LIN {X 0,Y 438.621,Z 496.858,A -85,B 0,C 180,E1 -9202.616,E2 -9202.616} C_VEL
LIN {X 0,Y 438.766,Z 492.887,A -85,B 0,C 180,E1 -9205.625,E2 -9205.625} C_VEL
LIN {X 0,Y 438.907,Z 491.24,A -85,B 0,C 180,E1 -9206.895,E2 -9206.895} C_VEL
LIN {X 0,Y 439.036,Z 496.514,A -85,B 0,C 180,E1 -9209.225,E2 -9209.225} C_VEL
LIN {X 0,Y 438.959,Z 503.716,A -85,B 0,C 180,E1 -9212.435,E2 -9212.435} C_VEL
LIN {X 0,Y 438.851,Z 509.893,A -85,B 0,C 180,E1 -9215.239,E2 -9215.239} C_VEL
LIN {X 0,Y 438.736,Z 517.378,A -85,B 0,C 180,E1 -9218.663,E2 -9218.663} C_VEL
LIN {X 0,Y 438.606,Z 523.965,A -85,B 0,C 180,E1 -9221.684,E2 -9221.684} C_VEL
LIN {X 0,Y 438.602,Z 527.103,A -85,B 0,C 180,E1 -9223.131,E2 -9223.131} C_VEL
LIN {X 0,Y 440.498,Z 538.596,A -85,B 0,C 180,E1 -9223.601,E2 -9223.601} C_VEL
LIN {X 0,Y 441.012,Z 543.733,A -85,B 0,C 180,E1 -9223.868,E2 -9223.868} C_VEL
LIN {X 0,Y 440.734,Z 552.93,A -85,B 0,C 180,E1 -9224.41,E2 -9224.41} C_VEL
LIN {X 0,Y 440.34,Z 561.813,A -85,B 0,C 180,E1 -9225.077,E2 -9225.077} C_VEL
LIN {X 0,Y 439.852,Z 572.155,A -85,B 0,C 180,E1 -9226.085,E2 -9226.085} C_VEL
LIN {X 0,Y 439.464,Z 579.635,A -85,B 0,C 180,E1 -9227.014,E2 -9227.014} C_VEL
LIN {X 0,Y 439.174,Z 584.756,A -85,B 0,C 180,E1 -9227.769,E2 -9227.769} C_VEL
LIN {X 0,Y 438.86,Z 590.657,A -85,B 0,C 180,E1 -9228.822,E2 -9228.822} C_VEL
LIN {X 0,Y 438.691,Z 595.327,A -85,B 0,C 180,E1 -9229.847,E2 -9229.847} C_VEL
LIN {X 0,Y 438.469,Z 600.506,A -85,B 0,C 180,E1 -9231.309,E2 -9231.309} C_VEL
LIN {X 0,Y 438.381,Z 603.477,A -85,B 0,C 180,E1 -9232.467,E2 -9232.467} C_VEL
LIN {X 0,Y 438.266,Z 605.527,A -85,B 0,C 180,E1 -9233.606,E2 -9233.606} C_VEL
LIN {X 0,Y 438.17,Z 606.89,A -85,B 0,C 180,E1 -9234.886,E2 -9234.886} C_VEL
LIN {X 0,Y 438.14,Z 607.23,A -85,B 0,C 180,E1 -9235.846,E2 -9235.846} C_VEL
LIN {X 0,Y 438.122,Z 606.973,A -85,B 0,C 180,E1 -9236.947,E2 -9236.947} C_VEL
LIN {X 0,Y 438.231,Z 605.831,A -85,B 0,C 180,E1 -9238.209,E2 -9238.209} C_VEL
LIN {X 0,Y 438.323,Z 604.322,A -85,B 0,C 180,E1 -9239.13,E2 -9239.13} C_VEL
LIN {X 0,Y 438.443,Z 600.496,A -85,B 0,C 180,E1 -9240.731,E2 -9240.731} C_VEL
LIN {X 0,Y 438.648,Z 595.849,A -85,B 0,C 180,E1 -9242.059,E2 -9242.059} C_VEL
LIN {X 0,Y 438.883,Z 591.19,A -85,B 0,C 180,E1 -9243.103,E2 -9243.103} C_VEL
LIN {X 0,Y 439.181,Z 584.982,A -85,B 0,C 180,E1 -9244.227,E2 -9244.227} C_VEL
LIN {X 0,Y 439.567,Z 576.57,A -85,B 0,C 180,E1 -9245.436,E2 -9245.436} C_VEL
LIN {X 0,Y 439.972,Z 568.448,A -85,B 0,C 180,E1 -9246.344,E2 -9246.344} C_VEL
LIN {X 0,Y 440.298,Z 560.08,A -85,B 0,C 180,E1 -9247.103,E2 -9247.103} C_VEL
LIN {X 0,Y 440.718,Z 550.964,A -85,B 0,C 180,E1 -9247.759,E2 -9247.759} C_VEL
LIN {X 0,Y 440.817,Z 542.35,A -85,B 0,C 180,E1 -9248.249,E2 -9248.249} C_VEL
LIN {X 0,Y 438.98,Z 530.4,A -85,B 0,C 180,E1 -9248.794,E2 -9248.794} C_VEL
LIN {X 0,Y 438.451,Z 527.192,A -85,B 0,C 180,E1 -9248.921,E2 -9248.921} C_VEL
LIN {X 0,Y 438.501,Z 521.905,A -85,B 0,C 180,E1 -9251.539,E2 -9251.539} C_VEL
LIN {X 0,Y 438.633,Z 516.526,A -85,B 0,C 180,E1 -9254.193,E2 -9254.193} C_VEL
LIN {X 0,Y 438.625,Z 514.073,A -85,B 0,C 180,E1 -9255.408,E2 -9255.408} C_VEL
LIN {X 0,Y 437.974,Z 512.647,A -85,B 0,C 180,E1 -9256.152,E2 -9256.152} C_VEL
LIN {X 0,Y 435.187,Z 510.501,A -85,B 0,C 180,E1 -9257.368,E2 -9257.368} C_VEL
LIN {X 0,Y 432.835,Z 508.797,A -85,B 0,C 180,E1 -9258.35,E2 -9258.35} C_VEL
LIN {X 0,Y 431.834,Z 507.335,A -85,B 0,C 180,E1 -9259.103,E2 -9259.103} C_VEL
LIN {X 0,Y 431.757,Z 506.816,A -85,B 0,C 180,E1 -9259.357,E2 -9259.357} C_VEL
LIN {X 0,Y 431.93,Z 499.414,A -85,B 0,C 180,E1 -9262.998,E2 -9262.998} C_VEL
LIN {X 0,Y 432.055,Z 494.709,A -85,B 0,C 180,E1 -9265.334,E2 -9265.334} C_VEL
LIN {X 0,Y 432.018,Z 491.487,A -85,B 0,C 180,E1 -9266.969,E2 -9266.969} C_VEL
LIN {X 0,Y 432.524,Z 491.421,A -85,B 0,C 180,E1 -9269.068,E2 -9269.068} C_VEL
LIN {X 0,Y 432.727,Z 491.397,A -85,B 0,C 180,E1 -9270,E2 -9270} C_VEL
LIN {X 0,Y 432.606,Z 491.412,A -85,B 0,C 180,E1 -9272.793,E2 -9272.793} C_VEL
LIN {X 0,Y 432.575,Z 491.416,A -85,B 0,C 180,E1 -9276.53,E2 -9276.53} C_VEL
LIN {X 0,Y 432.443,Z 491.429,A -85,B 0,C 180,E1 -9279.353,E2 -9279.353} C_VEL
LIN {X 0,Y 432.432,Z 491.432,A -85,B 0,C 180,E1 -9282.803,E2 -9282.803} C_VEL
LIN {X 0,Y 432.413,Z 491.436,A -85,B 0,C 180,E1 -9286.478,E2 -9286.478} C_VEL
LIN {X 0,Y 432.34,Z 491.445,A -85,B 0,C 180,E1 -9289.96,E2 -9289.96} C_VEL
LIN {X 0,Y 432.32,Z 491.446,A -85,B 0,C 180,E1 -9292.964,E2 -9292.964} C_VEL
LIN {X 0,Y 432.365,Z 491.442,A -85,B 0,C 180,E1 -9296.032,E2 -9296.032} C_VEL
LIN {X 0,Y 432.352,Z 491.441,A -85,B 0,C 180,E1 -9299.186,E2 -9299.186} C_VEL
LIN {X 0,Y 432.325,Z 491.449,A -85,B 0,C 180,E1 -9302.293,E2 -9302.293} C_VEL
LIN {X 0,Y 432.34,Z 491.444,A -85,B 0,C 180,E1 -9304.676,E2 -9304.676} C_VEL
LIN {X 0,Y 432.346,Z 491.445,A -85,B 0,C 180,E1 -9308.148,E2 -9308.148} C_VEL
LIN {X 0,Y 432.333,Z 491.445,A -85,B 0,C 180,E1 -9311.602,E2 -9311.602} C_VEL
LIN {X 0,Y 432.34,Z 491.445,A -85,B 0,C 180,E1 -9314.346,E2 -9314.346} C_VEL
LIN {X 0,Y 432.364,Z 491.439,A -85,B 0,C 180,E1 -9317.009,E2 -9317.009} C_VEL
LIN {X 0,Y 432.356,Z 491.443,A -85,B 0,C 180,E1 -9319.816,E2 -9319.816} C_VEL
LIN {X 0,Y 432.314,Z 491.445,A -85,B 0,C 180,E1 -9323.023,E2 -9323.023} C_VEL
LIN {X 0,Y 432.357,Z 491.445,A -85,B 0,C 180,E1 -9325.996,E2 -9325.996} C_VEL
LIN {X 0,Y 432.345,Z 491.443,A -85,B 0,C 180,E1 -9329.489,E2 -9329.489} C_VEL
LIN {X 0,Y 432.391,Z 491.437,A -85,B 0,C 180,E1 -9332.928,E2 -9332.928} C_VEL
LIN {X 0,Y 432.369,Z 491.442,A -85,B 0,C 180,E1 -9336.023,E2 -9336.023} C_VEL
LIN {X 0,Y 432.348,Z 491.442,A -85,B 0,C 180,E1 -9339.046,E2 -9339.046} C_VEL
LIN {X 0,Y 432.376,Z 491.441,A -85,B 0,C 180,E1 -9342.011,E2 -9342.011} C_VEL
LIN {X 0,Y 432.393,Z 491.437,A -85,B 0,C 180,E1 -9344.926,E2 -9344.926} C_VEL
LIN {X 0,Y 432.478,Z 491.428,A -85,B 0,C 180,E1 -9347.804,E2 -9347.804} C_VEL
LIN {X 0,Y 432.49,Z 491.426,A -85,B 0,C 180,E1 -9351.59,E2 -9351.59} C_VEL
LIN {X 0,Y 432.595,Z 491.412,A -85,B 0,C 180,E1 -9354.406,E2 -9354.406} C_VEL
LIN {X 0,Y 432.604,Z 491.412,A -85,B 0,C 180,E1 -9358.138,E2 -9358.138} C_VEL
LIN {X 0,Y 432.731,Z 491.397,A -85,B 0,C 180,E1 -9360,E2 -9360} C_VEL
LIN {X 0,Y 432.604,Z 491.41,A -85,B 0,C 180,E1 -9362.793,E2 -9362.793} C_VEL
LIN {X 0,Y 432.571,Z 491.414,A -85,B 0,C 180,E1 -9366.53,E2 -9366.53} C_VEL
LIN {X 0,Y 432.441,Z 491.432,A -85,B 0,C 180,E1 -9369.353,E2 -9369.353} C_VEL
LIN {X 0,Y 432.428,Z 491.431,A -85,B 0,C 180,E1 -9372.804,E2 -9372.804} C_VEL
LIN {X 0,Y 432.41,Z 491.435,A -85,B 0,C 180,E1 -9376.479,E2 -9376.479} C_VEL
LIN {X 0,Y 432.336,Z 491.446,A -85,B 0,C 180,E1 -9379.96,E2 -9379.96} C_VEL
LIN {X 0,Y 432.317,Z 491.447,A -85,B 0,C 180,E1 -9382.964,E2 -9382.964} C_VEL
LIN {X 0,Y 432.362,Z 491.443,A -85,B 0,C 180,E1 -9386.033,E2 -9386.033} C_VEL
LIN {X 0,Y 432.35,Z 491.444,A -85,B 0,C 180,E1 -9389.187,E2 -9389.187} C_VEL
LIN {X 0,Y 432.329,Z 491.445,A -85,B 0,C 180,E1 -9392.295,E2 -9392.295} C_VEL
LIN {X 0,Y 432.338,Z 491.444,A -85,B 0,C 180,E1 -9394.677,E2 -9394.677} C_VEL
LIN {X 0,Y 432.344,Z 491.443,A -85,B 0,C 180,E1 -9398.149,E2 -9398.149} C_VEL
LIN {X 0,Y 432.332,Z 491.448,A -85,B 0,C 180,E1 -9401.603,E2 -9401.603} C_VEL
LIN {X 0,Y 432.338,Z 491.443,A -85,B 0,C 180,E1 -9404.347,E2 -9404.347} C_VEL
LIN {X 0,Y 432.318,Z 491.447,A -85,B 0,C 180,E1 -9407.016,E2 -9407.016} C_VEL
LIN {X 0,Y 432.355,Z 491.443,A -85,B 0,C 180,E1 -9409.817,E2 -9409.817} C_VEL
LIN {X 0,Y 432.316,Z 491.449,A -85,B 0,C 180,E1 -9413.024,E2 -9413.024} C_VEL
LIN {X 0,Y 432.398,Z 491.49,A -85,B 0,C 180,E1 -9414.446,E2 -9414.446} C_VEL
LIN {X 0,Y 433.697,Z 498.9,A -85,B 0,C 180,E1 -9417.673,E2 -9417.673} C_VEL
LIN {X 0,Y 433.795,Z 502.505,A -85,B 0,C 180,E1 -9419.167,E2 -9419.167} C_VEL
LIN {X 0,Y 433.235,Z 510.767,A -85,B 0,C 180,E1 -9422.463,E2 -9422.463} C_VEL
LIN {X 0,Y 432.665,Z 519.988,A -85,B 0,C 180,E1 -9426.041,E2 -9426.041} C_VEL
LIN {X 0,Y 432.198,Z 529.205,A -85,B 0,C 180,E1 -9429.537,E2 -9429.537} C_VEL
LIN {X 0,Y 431.798,Z 538.416,A -85,B 0,C 180,E1 -9432.965,E2 -9432.965} C_VEL
LIN {X 0,Y 431.544,Z 547.609,A -85,B 0,C 180,E1 -9436.342,E2 -9436.342} C_VEL
LIN {X 0,Y 431.538,Z 549.403,A -85,B 0,C 180,E1 -9436.997,E2 -9436.997} C_VEL
LIN {X 0,Y 432.951,Z 563.611,A -85,B 0,C 180,E1 -9437.595,E2 -9437.595} C_VEL
LIN {X 0,Y 433.462,Z 570.117,A -85,B 0,C 180,E1 -9437.951,E2 -9437.951} C_VEL
LIN {X 0,Y 433.093,Z 580.396,A -85,B 0,C 180,E1 -9438.653,E2 -9438.653} C_VEL
LIN {X 0,Y 432.629,Z 589.892,A -85,B 0,C 180,E1 -9439.47,E2 -9439.47} C_VEL
LIN {X 0,Y 432.228,Z 598.533,A -85,B 0,C 180,E1 -9440.407,E2 -9440.407} C_VEL
LIN {X 0,Y 431.857,Z 607.082,A -85,B 0,C 180,E1 -9441.578,E2 -9441.578} C_VEL
LIN {X 0,Y 431.625,Z 613.803,A -85,B 0,C 180,E1 -9442.751,E2 -9442.751} C_VEL
LIN {X 0,Y 431.392,Z 618.953,A -85,B 0,C 180,E1 -9443.881,E2 -9443.881} C_VEL
LIN {X 0,Y 431.312,Z 623.981,A -85,B 0,C 180,E1 -9445.327,E2 -9445.327} C_VEL
LIN {X 0,Y 431.253,Z 626.448,A -85,B 0,C 180,E1 -9446.263,E2 -9446.263} C_VEL
LIN {X 0,Y 431.315,Z 628.342,A -85,B 0,C 180,E1 -9447.199,E2 -9447.199} C_VEL
LIN {X 0,Y 431.241,Z 629.637,A -85,B 0,C 180,E1 -9448.133,E2 -9448.133} C_VEL
LIN {X 0,Y 431.217,Z 630.481,A -85,B 0,C 180,E1 -9449.067,E2 -9449.067} C_VEL
LIN {X 0,Y 431.229,Z 630.751,A -85,B 0,C 180,E1 -9450,E2 -9450} C_VEL
LIN {X 0,Y 431.217,Z 630.501,A -85,B 0,C 180,E1 -9450.934,E2 -9450.934} C_VEL
LIN {X 0,Y 431.241,Z 629.661,A -85,B 0,C 180,E1 -9451.868,E2 -9451.868} C_VEL
LIN {X 0,Y 431.298,Z 628.374,A -85,B 0,C 180,E1 -9452.802,E2 -9452.802} C_VEL
LIN {X 0,Y 431.258,Z 625.37,A -85,B 0,C 180,E1 -9454.206,E2 -9454.206} C_VEL
LIN {X 0,Y 431.381,Z 621.08,A -85,B 0,C 180,E1 -9455.61,E2 -9455.61} C_VEL
LIN {X 0,Y 431.574,Z 615.227,A -85,B 0,C 180,E1 -9457.016,E2 -9457.016} C_VEL
LIN {X 0,Y 431.798,Z 608.9,A -85,B 0,C 180,E1 -9458.188,E2 -9458.188} C_VEL
LIN {X 0,Y 432.103,Z 602.762,A -85,B 0,C 180,E1 -9459.125,E2 -9459.125} C_VEL
LIN {X 0,Y 432.504,Z 595.348,A -85,B 0,C 180,E1 -9460.061,E2 -9460.061} C_VEL
LIN {X 0,Y 432.877,Z 587.491,A -85,B 0,C 180,E1 -9460.88,E2 -9460.88} C_VEL
LIN {X 0,Y 433.315,Z 579.319,A -85,B 0,C 180,E1 -9461.579,E2 -9461.579} C_VEL
LIN {X 0,Y 433.54,Z 569.525,A -85,B 0,C 180,E1 -9462.261,E2 -9462.261} C_VEL
LIN {X 0,Y 432.645,Z 557.327,A -85,B 0,C 180,E1 -9462.928,E2 -9462.928} C_VEL
LIN {X 0,Y 431.458,Z 548.071,A -85,B 0,C 180,E1 -9463.332,E2 -9463.332} C_VEL
LIN {X 0,Y 431.671,Z 539.83,A -85,B 0,C 180,E1 -9466.506,E2 -9466.506} C_VEL
LIN {X 0,Y 431.98,Z 531.096,A -85,B 0,C 180,E1 -9469.978,E2 -9469.978} C_VEL
LIN {X 0,Y 432.36,Z 522.72,A -85,B 0,C 180,E1 -9473.469,E2 -9473.469} C_VEL
LIN {X 0,Y 432.861,Z 515.354,A -85,B 0,C 180,E1 -9476.749,E2 -9476.749} C_VEL
LIN {X 0,Y 433.501,Z 508.305,A -85,B 0,C 180,E1 -9480.171,E2 -9480.171} C_VEL
LIN {X 0,Y 433.965,Z 503.76,A -85,B 0,C 180,E1 -9482.634,E2 -9482.634} C_VEL
LIN {X 0,Y 433.895,Z 500.697,A -85,B 0,C 180,E1 -9484.536,E2 -9484.536} C_VEL
LIN {X 0,Y 433.311,Z 496.888,A -85,B 0,C 180,E1 -9487.369,E2 -9487.369} C_VEL
LIN {X 0,Y 432.757,Z 493.7,A -85,B 0,C 180,E1 -9490.512,E2 -9490.512} C_VEL
LIN {X 0,Y 432.395,Z 491.961,A -85,B 0,C 180,E1 -9493.052,E2 -9493.052} C_VEL
LIN {X 0,Y 432.336,Z 491.447,A -85,B 0,C 180,E1 -9494.348,E2 -9494.348} C_VEL
LIN {X 0,Y 432.327,Z 491.448,A -85,B 0,C 180,E1 -9497.015,E2 -9497.015} C_VEL
LIN {X 0,Y 432.339,Z 491.446,A -85,B 0,C 180,E1 -9499.821,E2 -9499.821} C_VEL
LIN {X 0,Y 432.325,Z 491.563,A -85,B 0,C 180,E1 -9502.803,E2 -9502.803} C_VEL
LIN {X 0,Y 432.584,Z 493.097,A -85,B 0,C 180,E1 -9505.953,E2 -9505.953} C_VEL
LIN {X 0,Y 432.57,Z 494.889,A -85,B 0,C 180,E1 -9508.674,E2 -9508.674} C_VEL
LIN {X 0,Y 432.324,Z 497.455,A -85,B 0,C 180,E1 -9511.873,E2 -9511.873} C_VEL
LIN {X 0,Y 432.05,Z 500.247,A -85,B 0,C 180,E1 -9514.98,E2 -9514.98} C_VEL
LIN {X 0,Y 431.887,Z 503.238,A -85,B 0,C 180,E1 -9518.057,E2 -9518.057} C_VEL
LIN {X 0,Y 431.798,Z 506.271,A -85,B 0,C 180,E1 -9521.003,E2 -9521.003} C_VEL
LIN {X 0,Y 431.694,Z 509.44,A -85,B 0,C 180,E1 -9523.933,E2 -9523.933} C_VEL
LIN {X 0,Y 431.578,Z 512.837,A -85,B 0,C 180,E1 -9526.822,E2 -9526.822} C_VEL
LIN {X 0,Y 433.76,Z 522.586,A -85,B 0,C 180,E1 -9527.335,E2 -9527.335} C_VEL
LIN {X 0,Y 434.354,Z 528.796,A -85,B 0,C 180,E1 -9527.7,E2 -9527.7} C_VEL
LIN {X 0,Y 433.88,Z 539.519,A -85,B 0,C 180,E1 -9528.437,E2 -9528.437} C_VEL
LIN {X 0,Y 433.496,Z 547.554,A -85,B 0,C 180,E1 -9529.137,E2 -9529.137} C_VEL
LIN {X 0,Y 433.088,Z 555.269,A -85,B 0,C 180,E1 -9529.954,E2 -9529.954} C_VEL
LIN {X 0,Y 432.727,Z 562.542,A -85,B 0,C 180,E1 -9530.889,E2 -9530.889} C_VEL
LIN {X 0,Y 432.281,Z 569.949,A -85,B 0,C 180,E1 -9532.057,E2 -9532.057} C_VEL
LIN {X 0,Y 432.003,Z 576.748,A -85,B 0,C 180,E1 -9533.461,E2 -9533.461} C_VEL
LIN {X 0,Y 431.62,Z 580.395,A -85,B 0,C 180,E1 -9534.394,E2 -9534.394} C_VEL
LIN {X 0,Y 431.678,Z 583.344,A -85,B 0,C 180,E1 -9535.331,E2 -9535.331} C_VEL
LIN {X 0,Y 431.528,Z 585.637,A -85,B 0,C 180,E1 -9536.265,E2 -9536.265} C_VEL
LIN {X 0,Y 431.393,Z 587.351,A -85,B 0,C 180,E1 -9537.199,E2 -9537.199} C_VEL
LIN {X 0,Y 431.332,Z 588.555,A -85,B 0,C 180,E1 -9538.133,E2 -9538.133} C_VEL
LIN {X 0,Y 431.25,Z 589.276,A -85,B 0,C 180,E1 -9539.066,E2 -9539.066} C_VEL
LIN {X 0,Y 431.231,Z 589.505,A -85,B 0,C 180,E1 -9540,E2 -9540} C_VEL
LIN {X 0,Y 431.235,Z 589.141,A -85,B 0,C 180,E1 -9540.934,E2 -9540.934} C_VEL
LIN {X 0,Y 431.295,Z 588.253,A -85,B 0,C 180,E1 -9541.868,E2 -9541.868} C_VEL
LIN {X 0,Y 431.379,Z 586.874,A -85,B 0,C 180,E1 -9542.802,E2 -9542.802} C_VEL
LIN {X 0,Y 431.522,Z 583.791,A -85,B 0,C 180,E1 -9544.203,E2 -9544.203} C_VEL
LIN {X 0,Y 431.604,Z 579.415,A -85,B 0,C 180,E1 -9545.607,E2 -9545.607} C_VEL
LIN {X 0,Y 431.963,Z 574.673,A -85,B 0,C 180,E1 -9546.744,E2 -9546.744} C_VEL
LIN {X 0,Y 432.077,Z 568.326,A -85,B 0,C 180,E1 -9547.947,E2 -9547.947} C_VEL
LIN {X 0,Y 432.369,Z 562.276,A -85,B 0,C 180,E1 -9548.883,E2 -9548.883} C_VEL
LIN {X 0,Y 432.776,Z 553.923,A -85,B 0,C 180,E1 -9549.936,E2 -9549.936} C_VEL
LIN {X 0,Y 433.224,Z 544.72,A -85,B 0,C 180,E1 -9550.87,E2 -9550.87} C_VEL
LIN {X 0,Y 433.664,Z 534.251,A -85,B 0,C 180,E1 -9551.688,E2 -9551.688} C_VEL
LIN {X 0,Y 433.847,Z 525.581,A -85,B 0,C 180,E1 -9552.217,E2 -9552.217} C_VEL
LIN {X 0,Y 432.406,Z 516.149,A -85,B 0,C 180,E1 -9552.701,E2 -9552.701} C_VEL
LIN {X 0,Y 431.403,Z 510.563,A -85,B 0,C 180,E1 -9552.962,E2 -9552.962} C_VEL
LIN {X 0,Y 431.44,Z 506.27,A -85,B 0,C 180,E1 -9556.077,E2 -9556.077} C_VEL
LIN {X 0,Y 431.505,Z 502.098,A -85,B 0,C 180,E1 -9559.15,E2 -9559.15} C_VEL
LIN {X 0,Y 431.528,Z 498.31,A -85,B 0,C 180,E1 -9561.999,E2 -9561.999} C_VEL
LIN {X 0,Y 431.662,Z 494.317,A -85,B 0,C 180,E1 -9565.044,E2 -9565.044} C_VEL
LIN {X 0,Y 431.851,Z 492.008,A -85,B 0,C 180,E1 -9566.826,E2 -9566.826} C_VEL
LIN {X 0,Y 432.009,Z 495.847,A -85,B 0,C 180,E1 -9568.539,E2 -9568.539} C_VEL
LIN {X 0,Y 431.937,Z 502.183,A -85,B 0,C 180,E1 -9571.377,E2 -9571.377} C_VEL
LIN {X 0,Y 431.896,Z 507.785,A -85,B 0,C 180,E1 -9573.911,E2 -9573.911} C_VEL
LIN {X 0,Y 431.732,Z 514.698,A -85,B 0,C 180,E1 -9577.093,E2 -9577.093} C_VEL
LIN {X 0,Y 431.6,Z 521.116,A -85,B 0,C 180,E1 -9580.063,E2 -9580.063} C_VEL
LIN {X 0,Y 431.558,Z 527.411,A -85,B 0,C 180,E1 -9582.921,E2 -9582.921} C_VEL
LIN {X 0,Y 433.185,Z 537.127,A -85,B 0,C 180,E1 -9583.312,E2 -9583.312} C_VEL
LIN {X 0,Y 434.092,Z 544.931,A -85,B 0,C 180,E1 -9583.719,E2 -9583.719} C_VEL
LIN {X 0,Y 433.645,Z 556.12,A -85,B 0,C 180,E1 -9584.416,E2 -9584.416} C_VEL
LIN {X 0,Y 433.215,Z 565.628,A -85,B 0,C 180,E1 -9585.222,E2 -9585.222} C_VEL
LIN {X 0,Y 432.802,Z 573.348,A -85,B 0,C 180,E1 -9586.037,E2 -9586.037} C_VEL
LIN {X 0,Y 432.436,Z 580.464,A -85,B 0,C 180,E1 -9586.953,E2 -9586.953} C_VEL
LIN {X 0,Y 431.99,Z 588.079,A -85,B 0,C 180,E1 -9588.162,E2 -9588.162} C_VEL
LIN {X 0,Y 431.705,Z 594.036,A -85,B 0,C 180,E1 -9589.368,E2 -9589.368} C_VEL
LIN {X 0,Y 431.517,Z 598.612,A -85,B 0,C 180,E1 -9590.566,E2 -9590.566} C_VEL
LIN {X 0,Y 431.335,Z 602.092,A -85,B 0,C 180,E1 -9591.745,E2 -9591.745} C_VEL
LIN {X 0,Y 431.222,Z 604.77,A -85,B 0,C 180,E1 -9592.996,E2 -9592.996} C_VEL
LIN {X 0,Y 431.093,Z 606.849,A -85,B 0,C 180,E1 -9594.601,E2 -9594.601} C_VEL
LIN {X 0,Y 431.026,Z 607.379,A -85,B 0,C 180,E1 -9596.332,E2 -9596.332} C_VEL
LIN {X 0,Y 431.102,Z 606.298,A -85,B 0,C 180,E1 -9597.965,E2 -9597.965} C_VEL
LIN {X 0,Y 431.16,Z 605.558,A -85,B 0,C 180,E1 -9598.559,E2 -9598.559} C_VEL
LIN {X 0,Y 431.275,Z 603.398,A -85,B 0,C 180,E1 -9599.732,E2 -9599.732} C_VEL
LIN {X 0,Y 431.361,Z 600.878,A -85,B 0,C 180,E1 -9600.739,E2 -9600.739} C_VEL
LIN {X 0,Y 431.585,Z 596.296,A -85,B 0,C 180,E1 -9602.084,E2 -9602.084} C_VEL
LIN {X 0,Y 431.814,Z 591.248,A -85,B 0,C 180,E1 -9603.237,E2 -9603.237} C_VEL
LIN {X 0,Y 432.11,Z 586.005,A -85,B 0,C 180,E1 -9604.21,E2 -9604.21} C_VEL
LIN {X 0,Y 432.426,Z 578.906,A -85,B 0,C 180,E1 -9605.29,E2 -9605.29} C_VEL
LIN {X 0,Y 432.948,Z 569.283,A -85,B 0,C 180,E1 -9606.438,E2 -9606.438} C_VEL
LIN {X 0,Y 433.311,Z 560.916,A -85,B 0,C 180,E1 -9607.22,E2 -9607.22} C_VEL
LIN {X 0,Y 433.709,Z 552.639,A -85,B 0,C 180,E1 -9607.841,E2 -9607.841} C_VEL
LIN {X 0,Y 433.9,Z 543.655,A -85,B 0,C 180,E1 -9608.377,E2 -9608.377} C_VEL
LIN {X 0,Y 432.458,Z 533.788,A -85,B 0,C 180,E1 -9608.864,E2 -9608.864} C_VEL
LIN {X 0,Y 431.377,Z 527.349,A -85,B 0,C 180,E1 -9609.121,E2 -9609.121} C_VEL
LIN {X 0,Y 431.429,Z 521.633,A -85,B 0,C 180,E1 -9611.97,E2 -9611.97} C_VEL
LIN {X 0,Y 431.55,Z 515.753,A -85,B 0,C 180,E1 -9614.896,E2 -9614.896} C_VEL
LIN {X 0,Y 431.753,Z 510.04,A -85,B 0,C 180,E1 -9617.783,E2 -9617.783} C_VEL
LIN {X 0,Y 431.757,Z 506.816,A -85,B 0,C 180,E1 -9619.357,E2 -9619.357} C_VEL
LIN {X 0,Y 431.118,Z 505.356,A -85,B 0,C 180,E1 -9620.111,E2 -9620.111} C_VEL
LIN {X 0,Y 428.34,Z 503.182,A -85,B 0,C 180,E1 -9621.343,E2 -9621.343} C_VEL
LIN {X 0,Y 425.981,Z 501.433,A -85,B 0,C 180,E1 -9622.338,E2 -9622.338} C_VEL
LIN {X 0,Y 424.964,Z 499.976,A -85,B 0,C 180,E1 -9623.103,E2 -9623.103} C_VEL
LIN {X 0,Y 424.879,Z 499.459,A -85,B 0,C 180,E1 -9623.362,E2 -9623.362} C_VEL
LIN {X 0,Y 424.988,Z 495.672,A -85,B 0,C 180,E1 -9625.257,E2 -9625.257} C_VEL
LIN {X 0,Y 424.97,Z 492.365,A -85,B 0,C 180,E1 -9626.919,E2 -9626.919} C_VEL
LIN {X 0,Y 425.483,Z 492.298,A -85,B 0,C 180,E1 -9629.053,E2 -9629.053} C_VEL
LIN {X 0,Y 425.696,Z 492.272,A -85,B 0,C 180,E1 -9630,E2 -9630} C_VEL
LIN {X 0,Y 425.558,Z 492.289,A -85,B 0,C 180,E1 -9632.839,E2 -9632.839} C_VEL
LIN {X 0,Y 425.533,Z 492.293,A -85,B 0,C 180,E1 -9636.638,E2 -9636.638} C_VEL
LIN {X 0,Y 425.401,Z 492.307,A -85,B 0,C 180,E1 -9639.509,E2 -9639.509} C_VEL
LIN {X 0,Y 425.394,Z 492.309,A -85,B 0,C 180,E1 -9642.903,E2 -9642.903} C_VEL
LIN {X 0,Y 425.362,Z 492.315,A -85,B 0,C 180,E1 -9646.605,E2 -9646.605} C_VEL
LIN {X 0,Y 425.329,Z 492.317,A -85,B 0,C 180,E1 -9649.635,E2 -9649.635} C_VEL
LIN {X 0,Y 425.307,Z 492.319,A -85,B 0,C 180,E1 -9653.365,E2 -9653.365} C_VEL
LIN {X 0,Y 425.349,Z 492.314,A -85,B 0,C 180,E1 -9656.844,E2 -9656.844} C_VEL
LIN {X 0,Y 425.318,Z 492.319,A -85,B 0,C 180,E1 -9659.717,E2 -9659.717} C_VEL
LIN {X 0,Y 425.282,Z 492.321,A -85,B 0,C 180,E1 -9663.047,E2 -9663.047} C_VEL
LIN {X 0,Y 425.284,Z 492.325,A -85,B 0,C 180,E1 -9665.929,E2 -9665.929} C_VEL
LIN {X 0,Y 425.302,Z 492.319,A -85,B 0,C 180,E1 -9669.044,E2 -9669.044} C_VEL
LIN {X 0,Y 425.276,Z 492.324,A -85,B 0,C 180,E1 -9672.652,E2 -9672.652} C_VEL
LIN {X 0,Y 425.333,Z 492.318,A -85,B 0,C 180,E1 -9676.053,E2 -9676.053} C_VEL
LIN {X 0,Y 425.308,Z 492.32,A -85,B 0,C 180,E1 -9678.625,E2 -9678.625} C_VEL
LIN {X 0,Y 425.321,Z 492.317,A -85,B 0,C 180,E1 -9681.104,E2 -9681.104} C_VEL
LIN {X 0,Y 425.297,Z 492.321,A -85,B 0,C 180,E1 -9684.664,E2 -9684.664} C_VEL
LIN {X 0,Y 425.263,Z 492.327,A -85,B 0,C 180,E1 -9688.073,E2 -9688.073} C_VEL
LIN {X 0,Y 425.329,Z 492.317,A -85,B 0,C 180,E1 -9691.368,E2 -9691.368} C_VEL
LIN {X 0,Y 425.293,Z 492.32,A -85,B 0,C 180,E1 -9694.554,E2 -9694.554} C_VEL
LIN {X 0,Y 425.285,Z 492.324,A -85,B 0,C 180,E1 -9697.661,E2 -9697.661} C_VEL
LIN {X 0,Y 425.36,Z 492.312,A -85,B 0,C 180,E1 -9700.704,E2 -9700.704} C_VEL
LIN {X 0,Y 425.386,Z 492.312,A -85,B 0,C 180,E1 -9703.688,E2 -9703.688} C_VEL
LIN {X 0,Y 425.427,Z 492.307,A -85,B 0,C 180,E1 -9707.599,E2 -9707.599} C_VEL
LIN {X 0,Y 425.44,Z 492.304,A -85,B 0,C 180,E1 -9711.45,E2 -9711.45} C_VEL
LIN {X 0,Y 425.552,Z 492.29,A -85,B 0,C 180,E1 -9714.313,E2 -9714.313} C_VEL
LIN {X 0,Y 425.574,Z 492.288,A -85,B 0,C 180,E1 -9718.107,E2 -9718.107} C_VEL
LIN {X 0,Y 425.701,Z 492.273,A -85,B 0,C 180,E1 -9720,E2 -9720} C_VEL
LIN {X 0,Y 425.556,Z 492.288,A -85,B 0,C 180,E1 -9722.84,E2 -9722.84} C_VEL
LIN {X 0,Y 425.529,Z 492.29,A -85,B 0,C 180,E1 -9726.639,E2 -9726.639} C_VEL
LIN {X 0,Y 425.399,Z 492.31,A -85,B 0,C 180,E1 -9729.509,E2 -9729.509} C_VEL
LIN {X 0,Y 425.39,Z 492.308,A -85,B 0,C 180,E1 -9732.904,E2 -9732.904} C_VEL
LIN {X 0,Y 425.359,Z 492.313,A -85,B 0,C 180,E1 -9736.605,E2 -9736.605} C_VEL
LIN {X 0,Y 425.326,Z 492.319,A -85,B 0,C 180,E1 -9739.636,E2 -9739.636} C_VEL
LIN {X 0,Y 425.304,Z 492.322,A -85,B 0,C 180,E1 -9743.365,E2 -9743.365} C_VEL
LIN {X 0,Y 425.345,Z 492.314,A -85,B 0,C 180,E1 -9746.845,E2 -9746.845} C_VEL
LIN {X 0,Y 425.316,Z 492.322,A -85,B 0,C 180,E1 -9749.718,E2 -9749.718} C_VEL
LIN {X 0,Y 425.282,Z 492.323,A -85,B 0,C 180,E1 -9753.048,E2 -9753.048} C_VEL
LIN {X 0,Y 425.282,Z 492.324,A -85,B 0,C 180,E1 -9755.929,E2 -9755.929} C_VEL
LIN {X 0,Y 425.297,Z 492.321,A -85,B 0,C 180,E1 -9759.044,E2 -9759.044} C_VEL
LIN {X 0,Y 425.275,Z 492.323,A -85,B 0,C 180,E1 -9762.653,E2 -9762.653} C_VEL
LIN {X 0,Y 425.259,Z 492.327,A -85,B 0,C 180,E1 -9766.044,E2 -9766.044} C_VEL
LIN {X 0,Y 425.302,Z 492.319,A -85,B 0,C 180,E1 -9768.625,E2 -9768.625} C_VEL
LIN {X 0,Y 425.323,Z 492.319,A -85,B 0,C 180,E1 -9771.105,E2 -9771.105} C_VEL
LIN {X 0,Y 425.326,Z 492.364,A -85,B 0,C 180,E1 -9774.26,E2 -9774.26} C_VEL
LIN {X 0,Y 426.502,Z 498.913,A -85,B 0,C 180,E1 -9777.181,E2 -9777.181} C_VEL
LIN {X 0,Y 426.806,Z 502.947,A -85,B 0,C 180,E1 -9778.899,E2 -9778.899} C_VEL
LIN {X 0,Y 426.19,Z 511.815,A -85,B 0,C 180,E1 -9782.502,E2 -9782.502} C_VEL
LIN {X 0,Y 425.59,Z 521.01,A -85,B 0,C 180,E1 -9786.136,E2 -9786.136} C_VEL
LIN {X 0,Y 425.109,Z 530.204,A -85,B 0,C 180,E1 -9789.686,E2 -9789.686} C_VEL
LIN {X 0,Y 424.702,Z 539.392,A -85,B 0,C 180,E1 -9793.167,E2 -9793.167} C_VEL
LIN {X 0,Y 424.452,Z 548.562,A -85,B 0,C 180,E1 -9796.597,E2 -9796.597} C_VEL
LIN {X 0,Y 424.449,Z 549.161,A -85,B 0,C 180,E1 -9796.82,E2 -9796.82} C_VEL
LIN {X 0,Y 425.809,Z 562.59,A -85,B 0,C 180,E1 -9797.384,E2 -9797.384} C_VEL
LIN {X 0,Y 426.413,Z 571.11,A -85,B 0,C 180,E1 -9797.87,E2 -9797.87} C_VEL
LIN {X 0,Y 425.969,Z 582.807,A -85,B 0,C 180,E1 -9798.702,E2 -9798.702} C_VEL
LIN {X 0,Y 425.579,Z 591.92,A -85,B 0,C 180,E1 -9799.534,E2 -9799.534} C_VEL
LIN {X 0,Y 425.117,Z 600.149,A -85,B 0,C 180,E1 -9800.485,E2 -9800.485} C_VEL
LIN {X 0,Y 424.749,Z 608.271,A -85,B 0,C 180,E1 -9801.676,E2 -9801.676} C_VEL
LIN {X 0,Y 424.535,Z 614.711,A -85,B 0,C 180,E1 -9802.868,E2 -9802.868} C_VEL
LIN {X 0,Y 424.283,Z 620.698,A -85,B 0,C 180,E1 -9804.297,E2 -9804.297} C_VEL
LIN {X 0,Y 424.178,Z 625.048,A -85,B 0,C 180,E1 -9805.725,E2 -9805.725} C_VEL
LIN {X 0,Y 424.211,Z 628.059,A -85,B 0,C 180,E1 -9807.152,E2 -9807.152} C_VEL
LIN {X 0,Y 424.166,Z 629.332,A -85,B 0,C 180,E1 -9808.101,E2 -9808.101} C_VEL
LIN {X 0,Y 424.134,Z 630.165,A -85,B 0,C 180,E1 -9809.051,E2 -9809.051} C_VEL
LIN {X 0,Y 424.143,Z 630.436,A -85,B 0,C 180,E1 -9810,E2 -9810} C_VEL
LIN {X 0,Y 424.134,Z 630.172,A -85,B 0,C 180,E1 -9810.95,E2 -9810.95} C_VEL
LIN {X 0,Y 424.166,Z 629.393,A -85,B 0,C 180,E1 -9811.899,E2 -9811.899} C_VEL
LIN {X 0,Y 424.194,Z 628.131,A -85,B 0,C 180,E1 -9812.849,E2 -9812.849} C_VEL
LIN {X 0,Y 424.179,Z 625.138,A -85,B 0,C 180,E1 -9814.276,E2 -9814.276} C_VEL
LIN {X 0,Y 424.287,Z 620.844,A -85,B 0,C 180,E1 -9815.704,E2 -9815.704} C_VEL
LIN {X 0,Y 424.503,Z 615.018,A -85,B 0,C 180,E1 -9817.133,E2 -9817.133} C_VEL
LIN {X 0,Y 424.757,Z 608.719,A -85,B 0,C 180,E1 -9818.325,E2 -9818.325} C_VEL
LIN {X 0,Y 425.097,Z 602.609,A -85,B 0,C 180,E1 -9819.277,E2 -9819.277} C_VEL
LIN {X 0,Y 425.533,Z 594.24,A -85,B 0,C 180,E1 -9820.347,E2 -9820.347} C_VEL
LIN {X 0,Y 426.018,Z 585.092,A -85,B 0,C 180,E1 -9821.298,E2 -9821.298} C_VEL
LIN {X 0,Y 426.603,Z 574.881,A -85,B 0,C 180,E1 -9822.126,E2 -9822.126} C_VEL
LIN {X 0,Y 426.382,Z 567.056,A -85,B 0,C 180,E1 -9822.653,E2 -9822.653} C_VEL
LIN {X 0,Y 425.56,Z 556.121,A -85,B 0,C 180,E1 -9823.241,E2 -9823.241} C_VEL
LIN {X 0,Y 424.373,Z 547.668,A -85,B 0,C 180,E1 -9823.62,E2 -9823.62} C_VEL
LIN {X 0,Y 424.631,Z 539.518,A -85,B 0,C 180,E1 -9826.837,E2 -9826.837} C_VEL
LIN {X 0,Y 424.966,Z 530.979,A -85,B 0,C 180,E1 -9830.322,E2 -9830.322} C_VEL
LIN {X 0,Y 425.373,Z 522.711,A -85,B 0,C 180,E1 -9833.878,E2 -9833.878} C_VEL
LIN {X 0,Y 425.874,Z 515.948,A -85,B 0,C 180,E1 -9836.984,E2 -9836.984} C_VEL
LIN {X 0,Y 426.501,Z 509.555,A -85,B 0,C 180,E1 -9840.172,E2 -9840.172} C_VEL
LIN {X 0,Y 426.872,Z 506.578,A -85,B 0,C 180,E1 -9841.793,E2 -9841.793} C_VEL
LIN {X 0,Y 426.987,Z 502.892,A -85,B 0,C 180,E1 -9844.03,E2 -9844.03} C_VEL
LIN {X 0,Y 426.576,Z 499.634,A -85,B 0,C 180,E1 -9846.379,E2 -9846.379} C_VEL
LIN {X 0,Y 426.022,Z 496.516,A -85,B 0,C 180,E1 -9849.163,E2 -9849.163} C_VEL
LIN {X 0,Y 425.612,Z 494.198,A -85,B 0,C 180,E1 -9852.006,E2 -9852.006} C_VEL
LIN {X 0,Y 425.356,Z 492.815,A -85,B 0,C 180,E1 -9854.727,E2 -9854.727} C_VEL
LIN {X 0,Y 425.281,Z 492.325,A -85,B 0,C 180,E1 -9857.348,E2 -9857.348} C_VEL
LIN {X 0,Y 425.332,Z 492.446,A -85,B 0,C 180,E1 -9860.952,E2 -9860.952} C_VEL
LIN {X 0,Y 425.499,Z 493.765,A -85,B 0,C 180,E1 -9864.683,E2 -9864.683} C_VEL
LIN {X 0,Y 425.639,Z 495.249,A -85,B 0,C 180,E1 -9867.363,E2 -9867.363} C_VEL
LIN {X 0,Y 425.439,Z 497.33,A -85,B 0,C 180,E1 -9870.292,E2 -9870.292} C_VEL
LIN {X 0,Y 425.187,Z 499.967,A -85,B 0,C 180,E1 -9873.494,E2 -9873.494} C_VEL
LIN {X 0,Y 424.913,Z 502.818,A -85,B 0,C 180,E1 -9876.612,E2 -9876.612} C_VEL
LIN {X 0,Y 424.791,Z 505.807,A -85,B 0,C 180,E1 -9879.669,E2 -9879.669} C_VEL
LIN {X 0,Y 424.63,Z 508.922,A -85,B 0,C 180,E1 -9882.668,E2 -9882.668} C_VEL
LIN {X 0,Y 424.541,Z 512.131,A -85,B 0,C 180,E1 -9885.622,E2 -9885.622} C_VEL
LIN {X 0,Y 424.545,Z 513.342,A -85,B 0,C 180,E1 -9886.539,E2 -9886.539} C_VEL
LIN {X 0,Y 426.981,Z 523.992,A -85,B 0,C 180,E1 -9887.131,E2 -9887.131} C_VEL
LIN {X 0,Y 427.511,Z 530.186,A -85,B 0,C 180,E1 -9887.506,E2 -9887.506} C_VEL
LIN {X 0,Y 427.008,Z 540.544,A -85,B 0,C 180,E1 -9888.248,E2 -9888.248} C_VEL
LIN {X 0,Y 426.487,Z 549.65,A -85,B 0,C 180,E1 -9889.076,E2 -9889.076} C_VEL
LIN {X 0,Y 426.058,Z 558.047,A -85,B 0,C 180,E1 -9890.026,E2 -9890.026} C_VEL
LIN {X 0,Y 425.54,Z 566.391,A -85,B 0,C 180,E1 -9891.213,E2 -9891.213} C_VEL
LIN {X 0,Y 425.133,Z 572.949,A -85,B 0,C 180,E1 -9892.4,E2 -9892.4} C_VEL
LIN {X 0,Y 424.978,Z 577.262,A -85,B 0,C 180,E1 -9893.353,E2 -9893.353} C_VEL
LIN {X 0,Y 424.585,Z 580.88,A -85,B 0,C 180,E1 -9894.3,E2 -9894.3} C_VEL
LIN {X 0,Y 424.626,Z 583.814,A -85,B 0,C 180,E1 -9895.253,E2 -9895.253} C_VEL
LIN {X 0,Y 424.48,Z 586.096,A -85,B 0,C 180,E1 -9896.203,E2 -9896.203} C_VEL
LIN {X 0,Y 424.328,Z 587.783,A -85,B 0,C 180,E1 -9897.152,E2 -9897.152} C_VEL
LIN {X 0,Y 424.253,Z 588.959,A -85,B 0,C 180,E1 -9898.101,E2 -9898.101} C_VEL
LIN {X 0,Y 424.167,Z 589.648,A -85,B 0,C 180,E1 -9899.051,E2 -9899.051} C_VEL
LIN {X 0,Y 424.145,Z 589.852,A -85,B 0,C 180,E1 -9900,E2 -9900} C_VEL
LIN {X 0,Y 424.152,Z 589.474,A -85,B 0,C 180,E1 -9900.949,E2 -9900.949} C_VEL
LIN {X 0,Y 424.218,Z 588.551,A -85,B 0,C 180,E1 -9901.899,E2 -9901.899} C_VEL
LIN {X 0,Y 424.311,Z 587.134,A -85,B 0,C 180,E1 -9902.848,E2 -9902.848} C_VEL
LIN {X 0,Y 424.427,Z 584.005,A -85,B 0,C 180,E1 -9904.273,E2 -9904.273} C_VEL
LIN {X 0,Y 424.54,Z 579.562,A -85,B 0,C 180,E1 -9905.7,E2 -9905.7} C_VEL
LIN {X 0,Y 424.88,Z 573.878,A -85,B 0,C 180,E1 -9907.034,E2 -9907.034} C_VEL
LIN {X 0,Y 425.022,Z 568.333,A -85,B 0,C 180,E1 -9908.08,E2 -9908.08} C_VEL
LIN {X 0,Y 425.339,Z 562.219,A -85,B 0,C 180,E1 -9909.031,E2 -9909.031} C_VEL
LIN {X 0,Y 425.732,Z 554.817,A -85,B 0,C 180,E1 -9909.982,E2 -9909.982} C_VEL
LIN {X 0,Y 426.102,Z 546.949,A -85,B 0,C 180,E1 -9910.814,E2 -9910.814} C_VEL
LIN {X 0,Y 426.522,Z 537.246,A -85,B 0,C 180,E1 -9911.645,E2 -9911.645} C_VEL
LIN {X 0,Y 426.849,Z 526.137,A -85,B 0,C 180,E1 -9912.359,E2 -9912.359} C_VEL
LIN {X 0,Y 425.231,Z 516.088,A -85,B 0,C 180,E1 -9912.881,E2 -9912.881} C_VEL
LIN {X 0,Y 424.32,Z 510.857,A -85,B 0,C 180,E1 -9913.137,E2 -9913.137} C_VEL
LIN {X 0,Y 424.348,Z 506.458,A -85,B 0,C 180,E1 -9916.353,E2 -9916.353} C_VEL
LIN {X 0,Y 424.427,Z 502.446,A -85,B 0,C 180,E1 -9919.34,E2 -9919.34} C_VEL
LIN {X 0,Y 424.487,Z 498.442,A -85,B 0,C 180,E1 -9922.383,E2 -9922.383} C_VEL
LIN {X 0,Y 424.609,Z 494.407,A -85,B 0,C 180,E1 -9925.489,E2 -9925.489} C_VEL
LIN {X 0,Y 424.782,Z 492.863,A -85,B 0,C 180,E1 -9926.767,E2 -9926.767} C_VEL
LIN {X 0,Y 425.012,Z 495.83,A -85,B 0,C 180,E1 -9928.117,E2 -9928.117} C_VEL
LIN {X 0,Y 424.903,Z 503.075,A -85,B 0,C 180,E1 -9931.401,E2 -9931.401} C_VEL
LIN {X 0,Y 424.79,Z 509.279,A -85,B 0,C 180,E1 -9934.23,E2 -9934.23} C_VEL
LIN {X 0,Y 424.668,Z 516.146,A -85,B 0,C 180,E1 -9937.404,E2 -9937.404} C_VEL
LIN {X 0,Y 424.515,Z 522.555,A -85,B 0,C 180,E1 -9940.399,E2 -9940.399} C_VEL
LIN {X 0,Y 424.483,Z 527.631,A -85,B 0,C 180,E1 -9942.689,E2 -9942.689} C_VEL
LIN {X 0,Y 426.092,Z 536.826,A -85,B 0,C 180,E1 -9943.067,E2 -9943.067} C_VEL
LIN {X 0,Y 427.153,Z 544.655,A -85,B 0,C 180,E1 -9943.481,E2 -9943.481} C_VEL
LIN {X 0,Y 426.885,Z 553.248,A -85,B 0,C 180,E1 -9944.007,E2 -9944.007} C_VEL
LIN {X 0,Y 426.444,Z 562.256,A -85,B 0,C 180,E1 -9944.706,E2 -9944.706} C_VEL
LIN {X 0,Y 425.94,Z 571.683,A -85,B 0,C 180,E1 -9945.638,E2 -9945.638} C_VEL
LIN {X 0,Y 425.468,Z 579.462,A -85,B 0,C 180,E1 -9946.619,E2 -9946.619} C_VEL
LIN {X 0,Y 425.135,Z 585.519,A -85,B 0,C 180,E1 -9947.546,E2 -9947.546} C_VEL
LIN {X 0,Y 424.794,Z 591.02,A -85,B 0,C 180,E1 -9948.564,E2 -9948.564} C_VEL
LIN {X 0,Y 424.581,Z 595.569,A -85,B 0,C 180,E1 -9949.59,E2 -9949.59} C_VEL
LIN {X 0,Y 424.47,Z 598.59,A -85,B 0,C 180,E1 -9950.398,E2 -9950.398} C_VEL
LIN {X 0,Y 424.266,Z 602.261,A -85,B 0,C 180,E1 -9951.655,E2 -9951.655} C_VEL
LIN {X 0,Y 424.157,Z 604.545,A -85,B 0,C 180,E1 -9952.686,E2 -9952.686} C_VEL
LIN {X 0,Y 424.005,Z 606.786,A -85,B 0,C 180,E1 -9954.31,E2 -9954.31} C_VEL
LIN {X 0,Y 423.932,Z 607.65,A -85,B 0,C 180,E1 -9955.987,E2 -9955.987} C_VEL
LIN {X 0,Y 423.992,Z 606.768,A -85,B 0,C 180,E1 -9957.711,E2 -9957.711} C_VEL
LIN {X 0,Y 424.175,Z 604.23,A -85,B 0,C 180,E1 -9959.493,E2 -9959.493} C_VEL
LIN {X 0,Y 424.283,Z 601.25,A -85,B 0,C 180,E1 -9960.748,E2 -9960.748} C_VEL
LIN {X 0,Y 424.456,Z 597.644,A -85,B 0,C 180,E1 -9961.88,E2 -9961.88} C_VEL
LIN {X 0,Y 424.705,Z 592.418,A -85,B 0,C 180,E1 -9963.143,E2 -9963.143} C_VEL
LIN {X 0,Y 425.061,Z 586.534,A -85,B 0,C 180,E1 -9964.277,E2 -9964.277} C_VEL
LIN {X 0,Y 425.364,Z 580.712,A -85,B 0,C 180,E1 -9965.199,E2 -9965.199} C_VEL
LIN {X 0,Y 425.726,Z 573.505,A -85,B 0,C 180,E1 -9966.143,E2 -9966.143} C_VEL
LIN {X 0,Y 426.235,Z 564.619,A -85,B 0,C 180,E1 -9967.086,E2 -9967.086} C_VEL
LIN {X 0,Y 426.652,Z 555.216,A -85,B 0,C 180,E1 -9967.863,E2 -9967.863} C_VEL
LIN {X 0,Y 427.011,Z 545.922,A -85,B 0,C 180,E1 -9968.455,E2 -9968.455} C_VEL
LIN {X 0,Y 425.865,Z 536.901,A -85,B 0,C 180,E1 -9968.933,E2 -9968.933} C_VEL
LIN {X 0,Y 424.297,Z 527.496,A -85,B 0,C 180,E1 -9969.328,E2 -9969.328} C_VEL
LIN {X 0,Y 424.372,Z 522.855,A -85,B 0,C 180,E1 -9971.659,E2 -9971.659} C_VEL
LIN {X 0,Y 424.48,Z 516.926,A -85,B 0,C 180,E1 -9974.638,E2 -9974.638} C_VEL
LIN {X 0,Y 424.716,Z 509.112,A -85,B 0,C 180,E1 -9978.546,E2 -9978.546} C_VEL
LIN {X 0,Y 424.795,Z 503.418,A -85,B 0,C 180,E1 -9981.436,E2 -9981.436} C_VEL
LIN {X 0,Y 424.879,Z 499.459,A -85,B 0,C 180,E1 -9983.362,E2 -9983.362} C_VEL
LIN {X 0,Y 424.181,Z 498.034,A -85,B 0,C 180,E1 -9984.126,E2 -9984.126} C_VEL
LIN {X 0,Y 421.28,Z 495.858,A -85,B 0,C 180,E1 -9985.372,E2 -9985.372} C_VEL
LIN {X 0,Y 418.514,Z 493.763,A -85,B 0,C 180,E1 -9986.649,E2 -9986.649} C_VEL
LIN {X 0,Y 418.045,Z 493.225,A -85,B 0,C 180,E1 -9987.453,E2 -9987.453} C_VEL
LIN {X 0,Y 418.664,Z 493.148,A -85,B 0,C 180,E1 -9990,E2 -9990} C_VEL
LIN {X 0,Y 418.511,Z 493.166,A -85,B 0,C 180,E1 -9992.887,E2 -9992.887} C_VEL
LIN {X 0,Y 418.496,Z 493.168,A -85,B 0,C 180,E1 -9996.75,E2 -9996.75} C_VEL
LIN {X 0,Y 418.401,Z 493.181,A -85,B 0,C 180,E1 -9998.695,E2 -9998.695} C_VEL
LIN {X 0,Y 418.356,Z 493.186,A -85,B 0,C 180,E1 -10002.614,E2 -10002.614} C_VEL
LIN {X 0,Y 418.304,Z 493.191,A -85,B 0,C 180,E1 -10005.593,E2 -10005.593} C_VEL
LIN {X 0,Y 418.285,Z 493.195,A -85,B 0,C 180,E1 -10008.616,E2 -10008.616} C_VEL
LIN {X 0,Y 418.234,Z 493.2,A -85,B 0,C 180,E1 -10011.696,E2 -10011.696} C_VEL
LIN {X 0,Y 418.284,Z 493.194,A -85,B 0,C 180,E1 -10014.864,E2 -10014.864} C_VEL
LIN {X 0,Y 418.295,Z 493.195,A -85,B 0,C 180,E1 -10018.062,E2 -10018.062} C_VEL
LIN {X 0,Y 418.216,Z 493.203,A -85,B 0,C 180,E1 -10021.395,E2 -10021.395} C_VEL
LIN {X 0,Y 418.265,Z 493.198,A -85,B 0,C 180,E1 -10024.58,E2 -10024.58} C_VEL
LIN {X 0,Y 418.234,Z 493.202,A -85,B 0,C 180,E1 -10027.834,E2 -10027.834} C_VEL
LIN {X 0,Y 418.222,Z 493.201,A -85,B 0,C 180,E1 -10030.947,E2 -10030.947} C_VEL
LIN {X 0,Y 418.215,Z 493.204,A -85,B 0,C 180,E1 -10033.73,E2 -10033.73} C_VEL
LIN {X 0,Y 418.282,Z 493.196,A -85,B 0,C 180,E1 -10036.458,E2 -10036.458} C_VEL
LIN {X 0,Y 418.265,Z 493.196,A -85,B 0,C 180,E1 -10039.123,E2 -10039.123} C_VEL
LIN {X 0,Y 418.236,Z 493.203,A -85,B 0,C 180,E1 -10042.164,E2 -10042.164} C_VEL
LIN {X 0,Y 418.263,Z 493.198,A -85,B 0,C 180,E1 -10045.419,E2 -10045.419} C_VEL
LIN {X 0,Y 418.209,Z 493.203,A -85,B 0,C 180,E1 -10048.604,E2 -10048.604} C_VEL
LIN {X 0,Y 418.29,Z 493.197,A -85,B 0,C 180,E1 -10051.936,E2 -10051.936} C_VEL
LIN {X 0,Y 418.287,Z 493.192,A -85,B 0,C 180,E1 -10055.162,E2 -10055.162} C_VEL
LIN {X 0,Y 418.232,Z 493.202,A -85,B 0,C 180,E1 -10058.303,E2 -10058.303} C_VEL
LIN {X 0,Y 418.281,Z 493.195,A -85,B 0,C 180,E1 -10061.383,E2 -10061.383} C_VEL
LIN {X 0,Y 418.3,Z 493.193,A -85,B 0,C 180,E1 -10064.406,E2 -10064.406} C_VEL
LIN {X 0,Y 418.368,Z 493.185,A -85,B 0,C 180,E1 -10067.386,E2 -10067.386} C_VEL
LIN {X 0,Y 418.357,Z 493.186,A -85,B 0,C 180,E1 -10070.329,E2 -10070.329} C_VEL
LIN {X 0,Y 418.491,Z 493.169,A -85,B 0,C 180,E1 -10073.249,E2 -10073.249} C_VEL
LIN {X 0,Y 418.339,Z 493.187,A -85,B 0,C 180,E1 -10075.181,E2 -10075.181} C_VEL
LIN {X 0,Y 418.543,Z 493.164,A -85,B 0,C 180,E1 -10078.075,E2 -10078.075} C_VEL
LIN {X 0,Y 418.67,Z 493.149,A -85,B 0,C 180,E1 -10080,E2 -10080} C_VEL
LIN {X 0,Y 418.51,Z 493.166,A -85,B 0,C 180,E1 -10082.888,E2 -10082.888} C_VEL
LIN {X 0,Y 418.492,Z 493.167,A -85,B 0,C 180,E1 -10086.751,E2 -10086.751} C_VEL
LIN {X 0,Y 418.355,Z 493.188,A -85,B 0,C 180,E1 -10089.671,E2 -10089.671} C_VEL
LIN {X 0,Y 418.343,Z 493.186,A -85,B 0,C 180,E1 -10093.001,E2 -10093.001} C_VEL
LIN {X 0,Y 418.31,Z 493.19,A -85,B 0,C 180,E1 -10096.736,E2 -10096.736} C_VEL
LIN {X 0,Y 418.268,Z 493.198,A -85,B 0,C 180,E1 -10099.791,E2 -10099.791} C_VEL
LIN {X 0,Y 418.235,Z 493.2,A -85,B 0,C 180,E1 -10102.736,E2 -10102.736} C_VEL
LIN {X 0,Y 418.268,Z 493.199,A -85,B 0,C 180,E1 -10105.904,E2 -10105.904} C_VEL
LIN {X 0,Y 418.272,Z 493.198,A -85,B 0,C 180,E1 -10109.161,E2 -10109.161} C_VEL
LIN {X 0,Y 418.258,Z 493.197,A -85,B 0,C 180,E1 -10112.845,E2 -10112.845} C_VEL
LIN {X 0,Y 418.246,Z 493.199,A -85,B 0,C 180,E1 -10116.239,E2 -10116.239} C_VEL
LIN {X 0,Y 418.249,Z 493.2,A -85,B 0,C 180,E1 -10119.682,E2 -10119.682} C_VEL
LIN {X 0,Y 418.23,Z 493.2,A -85,B 0,C 180,E1 -10122.322,E2 -10122.322} C_VEL
LIN {X 0,Y 418.235,Z 493.201,A -85,B 0,C 180,E1 -10125.109,E2 -10125.109} C_VEL
LIN {X 0,Y 418.254,Z 493.199,A -85,B 0,C 180,E1 -10127.769,E2 -10127.769} C_VEL
LIN {X 0,Y 418.267,Z 493.195,A -85,B 0,C 180,E1 -10130.617,E2 -10130.617} C_VEL
LIN {X 0,Y 418.296,Z 493.332,A -85,B 0,C 180,E1 -10134.13,E2 -10134.13} C_VEL
LIN {X 0,Y 419.395,Z 499.459,A -85,B 0,C 180,E1 -10136.916,E2 -10136.916} C_VEL
LIN {X 0,Y 419.788,Z 503.639,A -85,B 0,C 180,E1 -10138.736,E2 -10138.736} C_VEL
LIN {X 0,Y 419.225,Z 511.52,A -85,B 0,C 180,E1 -10142.005,E2 -10142.005} C_VEL
LIN {X 0,Y 418.648,Z 519.391,A -85,B 0,C 180,E1 -10145.186,E2 -10145.186} C_VEL
LIN {X 0,Y 418.211,Z 527.25,A -85,B 0,C 180,E1 -10148.303,E2 -10148.303} C_VEL
LIN {X 0,Y 417.825,Z 535.107,A -85,B 0,C 180,E1 -10151.363,E2 -10151.363} C_VEL
LIN {X 0,Y 417.505,Z 544.237,A -85,B 0,C 180,E1 -10154.876,E2 -10154.876} C_VEL
LIN {X 0,Y 417.367,Z 548.885,A -85,B 0,C 180,E1 -10156.647,E2 -10156.647} C_VEL
LIN {X 0,Y 418.687,Z 561.888,A -85,B 0,C 180,E1 -10157.195,E2 -10157.195} C_VEL
LIN {X 0,Y 419.385,Z 572.366,A -85,B 0,C 180,E1 -10157.786,E2 -10157.786} C_VEL
LIN {X 0,Y 419.04,Z 580.944,A -85,B 0,C 180,E1 -10158.39,E2 -10158.39} C_VEL
LIN {X 0,Y 418.64,Z 589.153,A -85,B 0,C 180,E1 -10159.114,E2 -10159.114} C_VEL
LIN {X 0,Y 418.272,Z 596.927,A -85,B 0,C 180,E1 -10159.961,E2 -10159.961} C_VEL
LIN {X 0,Y 417.857,Z 605.028,A -85,B 0,C 180,E1 -10161.05,E2 -10161.05} C_VEL
LIN {X 0,Y 417.517,Z 612.097,A -85,B 0,C 180,E1 -10162.261,E2 -10162.261} C_VEL
LIN {X 0,Y 417.255,Z 618.146,A -85,B 0,C 180,E1 -10163.596,E2 -10163.596} C_VEL
LIN {X 0,Y 417.198,Z 622.047,A -85,B 0,C 180,E1 -10164.684,E2 -10164.684} C_VEL
LIN {X 0,Y 417.069,Z 625.976,A -85,B 0,C 180,E1 -10166.136,E2 -10166.136} C_VEL
LIN {X 0,Y 417.106,Z 627.824,A -85,B 0,C 180,E1 -10167.103,E2 -10167.103} C_VEL
LIN {X 0,Y 417.093,Z 629.146,A -85,B 0,C 180,E1 -10168.069,E2 -10168.069} C_VEL
LIN {X 0,Y 417.054,Z 629.965,A -85,B 0,C 180,E1 -10169.035,E2 -10169.035} C_VEL
LIN {X 0,Y 417.059,Z 630.242,A -85,B 0,C 180,E1 -10170,E2 -10170} C_VEL
LIN {X 0,Y 417.054,Z 629.98,A -85,B 0,C 180,E1 -10170.966,E2 -10170.966} C_VEL
LIN {X 0,Y 417.093,Z 629.188,A -85,B 0,C 180,E1 -10171.932,E2 -10171.932} C_VEL
LIN {X 0,Y 417.09,Z 627.911,A -85,B 0,C 180,E1 -10172.898,E2 -10172.898} C_VEL
LIN {X 0,Y 417.105,Z 624.937,A -85,B 0,C 180,E1 -10174.349,E2 -10174.349} C_VEL
LIN {X 0,Y 417.2,Z 620.654,A -85,B 0,C 180,E1 -10175.801,E2 -10175.801} C_VEL
LIN {X 0,Y 417.445,Z 614.828,A -85,B 0,C 180,E1 -10177.254,E2 -10177.254} C_VEL
LIN {X 0,Y 417.73,Z 608.601,A -85,B 0,C 180,E1 -10178.466,E2 -10178.466} C_VEL
LIN {X 0,Y 418.084,Z 602.574,A -85,B 0,C 180,E1 -10179.434,E2 -10179.434} C_VEL
LIN {X 0,Y 418.515,Z 595.308,A -85,B 0,C 180,E1 -10180.401,E2 -10180.401} C_VEL
LIN {X 0,Y 418.952,Z 587.649,A -85,B 0,C 180,E1 -10181.246,E2 -10181.246} C_VEL
LIN {X 0,Y 419.434,Z 579.737,A -85,B 0,C 180,E1 -10181.968,E2 -10181.968} C_VEL
LIN {X 0,Y 419.733,Z 571.748,A -85,B 0,C 180,E1 -10182.573,E2 -10182.573} C_VEL
LIN {X 0,Y 419.133,Z 561.72,A -85,B 0,C 180,E1 -10183.212,E2 -10183.212} C_VEL
LIN {X 0,Y 417.664,Z 549.509,A -85,B 0,C 180,E1 -10183.832,E2 -10183.832} C_VEL
LIN {X 0,Y 417.321,Z 547.228,A -85,B 0,C 180,E1 -10183.948,E2 -10183.948} C_VEL
LIN {X 0,Y 417.581,Z 539.358,A -85,B 0,C 180,E1 -10187.13,E2 -10187.13} C_VEL
LIN {X 0,Y 417.929,Z 530.896,A -85,B 0,C 180,E1 -10190.68,E2 -10190.68} C_VEL
LIN {X 0,Y 418.389,Z 522.72,A -85,B 0,C 180,E1 -10194.302,E2 -10194.302} C_VEL
LIN {X 0,Y 418.882,Z 516.56,A -85,B 0,C 180,E1 -10197.223,E2 -10197.223} C_VEL
LIN {X 0,Y 419.519,Z 510.825,A -85,B 0,C 180,E1 -10200.171,E2 -10200.171} C_VEL
LIN {X 0,Y 419.936,Z 506.918,A -85,B 0,C 180,E1 -10202.382,E2 -10202.382} C_VEL
LIN {X 0,Y 419.99,Z 503.367,A -85,B 0,C 180,E1 -10204.677,E2 -10204.677} C_VEL
LIN {X 0,Y 419.498,Z 500.283,A -85,B 0,C 180,E1 -10207.094,E2 -10207.094} C_VEL
LIN {X 0,Y 419.055,Z 497.693,A -85,B 0,C 180,E1 -10209.591,E2 -10209.591} C_VEL
LIN {X 0,Y 418.663,Z 495.569,A -85,B 0,C 180,E1 -10212.386,E2 -10212.386} C_VEL
LIN {X 0,Y 418.431,Z 494.275,A -85,B 0,C 180,E1 -10215.135,E2 -10215.135} C_VEL
LIN {X 0,Y 418.342,Z 493.753,A -85,B 0,C 180,E1 -10217.78,E2 -10217.78} C_VEL
LIN {X 0,Y 418.358,Z 493.879,A -85,B 0,C 180,E1 -10220.603,E2 -10220.603} C_VEL
LIN {X 0,Y 418.501,Z 494.85,A -85,B 0,C 180,E1 -10224.002,E2 -10224.002} C_VEL
LIN {X 0,Y 418.651,Z 496.367,A -85,B 0,C 180,E1 -10227.074,E2 -10227.074} C_VEL
LIN {X 0,Y 418.491,Z 498.137,A -85,B 0,C 180,E1 -10229.748,E2 -10229.748} C_VEL
LIN {X 0,Y 418.195,Z 500.673,A -85,B 0,C 180,E1 -10233.016,E2 -10233.016} C_VEL
LIN {X 0,Y 417.918,Z 503.456,A -85,B 0,C 180,E1 -10236.197,E2 -10236.197} C_VEL
LIN {X 0,Y 417.771,Z 506.408,A -85,B 0,C 180,E1 -10239.312,E2 -10239.312} C_VEL
LIN {X 0,Y 417.609,Z 509.49,A -85,B 0,C 180,E1 -10242.367,E2 -10242.367} C_VEL
LIN {X 0,Y 417.505,Z 512.675,A -85,B 0,C 180,E1 -10245.375,E2 -10245.375} C_VEL
LIN {X 0,Y 417.504,Z 513.586,A -85,B 0,C 180,E1 -10246.214,E2 -10246.214} C_VEL
LIN {X 0,Y 420.081,Z 524.747,A -85,B 0,C 180,E1 -10246.866,E2 -10246.866} C_VEL
LIN {X 0,Y 420.729,Z 530.309,A -85,B 0,C 180,E1 -10247.222,E2 -10247.222} C_VEL
LIN {X 0,Y 420.207,Z 540.154,A -85,B 0,C 180,E1 -10247.933,E2 -10247.933} C_VEL
LIN {X 0,Y 419.661,Z 549.373,A -85,B 0,C 180,E1 -10248.774,E2 -10248.774} C_VEL
LIN {X 0,Y 419.239,Z 556.89,A -85,B 0,C 180,E1 -10249.618,E2 -10249.618} C_VEL
LIN {X 0,Y 418.818,Z 563.988,A -85,B 0,C 180,E1 -10250.584,E2 -10250.584} C_VEL
LIN {X 0,Y 418.32,Z 571.235,A -85,B 0,C 180,E1 -10251.79,E2 -10251.79} C_VEL
LIN {X 0,Y 417.957,Z 577.857,A -85,B 0,C 180,E1 -10253.24,E2 -10253.24} C_VEL
LIN {X 0,Y 417.519,Z 582.908,A -85,B 0,C 180,E1 -10254.688,E2 -10254.688} C_VEL
LIN {X 0,Y 417.51,Z 585.44,A -85,B 0,C 180,E1 -10255.656,E2 -10255.656} C_VEL
LIN {X 0,Y 417.266,Z 588.22,A -85,B 0,C 180,E1 -10257.104,E2 -10257.104} C_VEL
LIN {X 0,Y 417.177,Z 589.36,A -85,B 0,C 180,E1 -10258.069,E2 -10258.069} C_VEL
LIN {X 0,Y 417.086,Z 590.019,A -85,B 0,C 180,E1 -10259.035,E2 -10259.035} C_VEL
LIN {X 0,Y 417.062,Z 590.194,A -85,B 0,C 180,E1 -10260,E2 -10260} C_VEL
LIN {X 0,Y 417.072,Z 589.805,A -85,B 0,C 180,E1 -10260.966,E2 -10260.966} C_VEL
LIN {X 0,Y 417.144,Z 588.844,A -85,B 0,C 180,E1 -10261.931,E2 -10261.931} C_VEL
LIN {X 0,Y 417.246,Z 587.388,A -85,B 0,C 180,E1 -10262.897,E2 -10262.897} C_VEL
LIN {X 0,Y 417.333,Z 584.212,A -85,B 0,C 180,E1 -10264.346,E2 -10264.346} C_VEL
LIN {X 0,Y 417.482,Z 579.697,A -85,B 0,C 180,E1 -10265.797,E2 -10265.797} C_VEL
LIN {X 0,Y 417.816,Z 574.427,A -85,B 0,C 180,E1 -10267.053,E2 -10267.053} C_VEL
LIN {X 0,Y 417.988,Z 568.324,A -85,B 0,C 180,E1 -10268.217,E2 -10268.217} C_VEL
LIN {X 0,Y 418.305,Z 562.138,A -85,B 0,C 180,E1 -10269.184,E2 -10269.184} C_VEL
LIN {X 0,Y 418.704,Z 554.653,A -85,B 0,C 180,E1 -10270.151,E2 -10270.151} C_VEL
LIN {X 0,Y 419.191,Z 545.478,A -85,B 0,C 180,E1 -10271.117,E2 -10271.117} C_VEL
LIN {X 0,Y 419.673,Z 535.102,A -85,B 0,C 180,E1 -10271.961,E2 -10271.961} C_VEL
LIN {X 0,Y 419.79,Z 526.542,A -85,B 0,C 180,E1 -10272.509,E2 -10272.509} C_VEL
LIN {X 0,Y 418.132,Z 516.355,A -85,B 0,C 180,E1 -10273.051,E2 -10273.051} C_VEL
LIN {X 0,Y 417.242,Z 511.156,A -85,B 0,C 180,E1 -10273.307,E2 -10273.307} C_VEL
LIN {X 0,Y 417.265,Z 506.646,A -85,B 0,C 180,E1 -10276.639,E2 -10276.639} C_VEL
LIN {X 0,Y 417.339,Z 502.596,A -85,B 0,C 180,E1 -10279.682,E2 -10279.682} C_VEL
LIN {X 0,Y 417.435,Z 498.559,A -85,B 0,C 180,E1 -10282.782,E2 -10282.782} C_VEL
LIN {X 0,Y 417.701,Z 493.645,A -85,B 0,C 180,E1 -10286.683,E2 -10286.683} C_VEL
LIN {X 0,Y 417.977,Z 496.709,A -85,B 0,C 180,E1 -10288.086,E2 -10288.086} C_VEL
LIN {X 0,Y 417.858,Z 503.981,A -85,B 0,C 180,E1 -10291.426,E2 -10291.426} C_VEL
LIN {X 0,Y 417.723,Z 510.598,A -85,B 0,C 180,E1 -10294.471,E2 -10294.471} C_VEL
LIN {X 0,Y 417.605,Z 517.592,A -85,B 0,C 180,E1 -10297.722,E2 -10297.722} C_VEL
LIN {X 0,Y 417.421,Z 524.645,A -85,B 0,C 180,E1 -10301.044,E2 -10301.044} C_VEL
LIN {X 0,Y 417.409,Z 527.595,A -85,B 0,C 180,E1 -10302.439,E2 -10302.439} C_VEL
LIN {X 0,Y 419.129,Z 537.446,A -85,B 0,C 180,E1 -10302.856,E2 -10302.856} C_VEL
LIN {X 0,Y 420.221,Z 545.397,A -85,B 0,C 180,E1 -10303.291,E2 -10303.291} C_VEL
LIN {X 0,Y 419.94,Z 553.915,A -85,B 0,C 180,E1 -10303.829,E2 -10303.829} C_VEL
LIN {X 0,Y 419.452,Z 563.561,A -85,B 0,C 180,E1 -10304.601,E2 -10304.601} C_VEL
LIN {X 0,Y 418.903,Z 573.307,A -85,B 0,C 180,E1 -10305.63,E2 -10305.63} C_VEL
LIN {X 0,Y 418.453,Z 579.853,A -85,B 0,C 180,E1 -10306.48,E2 -10306.48} C_VEL
LIN {X 0,Y 418.119,Z 585.898,A -85,B 0,C 180,E1 -10307.426,E2 -10307.426} C_VEL
LIN {X 0,Y 417.792,Z 590.889,A -85,B 0,C 180,E1 -10308.359,E2 -10308.359} C_VEL
LIN {X 0,Y 417.585,Z 594.843,A -85,B 0,C 180,E1 -10309.232,E2 -10309.232} C_VEL
LIN {X 0,Y 417.407,Z 598.567,A -85,B 0,C 180,E1 -10310.221,E2 -10310.221} C_VEL
LIN {X 0,Y 417.202,Z 602.159,A -85,B 0,C 180,E1 -10311.443,E2 -10311.443} C_VEL
LIN {X 0,Y 417.078,Z 604.796,A -85,B 0,C 180,E1 -10312.654,E2 -10312.654} C_VEL
LIN {X 0,Y 416.937,Z 606.725,A -85,B 0,C 180,E1 -10314.008,E2 -10314.008} C_VEL
LIN {X 0,Y 416.886,Z 607.557,A -85,B 0,C 180,E1 -10315.027,E2 -10315.027} C_VEL
LIN {X 0,Y 416.849,Z 607.804,A -85,B 0,C 180,E1 -10316.194,E2 -10316.194} C_VEL
LIN {X 0,Y 416.894,Z 607.234,A -85,B 0,C 180,E1 -10317.448,E2 -10317.448} C_VEL
LIN {X 0,Y 416.972,Z 606.138,A -85,B 0,C 180,E1 -10318.499,E2 -10318.499} C_VEL
LIN {X 0,Y 417.103,Z 604.23,A -85,B 0,C 180,E1 -10319.636,E2 -10319.636} C_VEL
LIN {X 0,Y 417.243,Z 600.416,A -85,B 0,C 180,E1 -10321.15,E2 -10321.15} C_VEL
LIN {X 0,Y 417.499,Z 596.061,A -85,B 0,C 180,E1 -10322.424,E2 -10322.424} C_VEL
LIN {X 0,Y 417.748,Z 590.976,A -85,B 0,C 180,E1 -10323.594,E2 -10323.594} C_VEL
LIN {X 0,Y 418.176,Z 583.755,A -85,B 0,C 180,E1 -10324.916,E2 -10324.916} C_VEL
LIN {X 0,Y 418.615,Z 575.261,A -85,B 0,C 180,E1 -10326.107,E2 -10326.107} C_VEL
LIN {X 0,Y 419.072,Z 567.974,A -85,B 0,C 180,E1 -10326.933,E2 -10326.933} C_VEL
LIN {X 0,Y 419.367,Z 561.069,A -85,B 0,C 180,E1 -10327.588,E2 -10327.588} C_VEL
LIN {X 0,Y 419.851,Z 552.255,A -85,B 0,C 180,E1 -10328.262,E2 -10328.262} C_VEL
LIN {X 0,Y 419.947,Z 544.898,A -85,B 0,C 180,E1 -10328.718,E2 -10328.718} C_VEL
LIN {X 0,Y 418.521,Z 535.3,A -85,B 0,C 180,E1 -10329.222,E2 -10329.222} C_VEL
LIN {X 0,Y 417.222,Z 527.647,A -85,B 0,C 180,E1 -10329.541,E2 -10329.541} C_VEL
LIN {X 0,Y 417.332,Z 521.09,A -85,B 0,C 180,E1 -10332.86,E2 -10332.86} C_VEL
LIN {X 0,Y 417.415,Z 516.117,A -85,B 0,C 180,E1 -10335.371,E2 -10335.371} C_VEL
LIN {X 0,Y 417.657,Z 510.238,A -85,B 0,C 180,E1 -10338.35,E2 -10338.35} C_VEL
LIN {X 0,Y 417.728,Z 504.449,A -85,B 0,C 180,E1 -10341.29,E2 -10341.29} C_VEL
LIN {X 0,Y 417.844,Z 498.584,A -85,B 0,C 180,E1 -10344.207,E2 -10344.207} C_VEL
LIN {X 0,Y 417.933,Z 493.242,A -85,B 0,C 180,E1 -10346.927,E2 -10346.927} C_VEL
LIN {X 0,Y 418.045,Z 493.225,A -85,B 0,C 180,E1 -10347.453,E2 -10347.453} C_VEL
LIN {X 0,Y 417.59,Z 493.284,A -85,B 0,C 180,E1 -10348.26,E2 -10348.26} C_VEL
LIN {X 0,Y 414.905,Z 493.615,A -85,B 0,C 180,E1 -10349.576,E2 -10349.576} C_VEL
LIN {X 0,Y 412.543,Z 493.911,A -85,B 0,C 180,E1 -10350.638,E2 -10350.638} C_VEL
LIN {X 0,Y 411.554,Z 494.032,A -85,B 0,C 180,E1 -10351.458,E2 -10351.458} C_VEL
LIN {X 0,Y 411.493,Z 494.04,A -85,B 0,C 180,E1 -10351.735,E2 -10351.735} C_VEL
LIN {X 0,Y 411.478,Z 494.043,A -85,B 0,C 180,E1 -10355.881,E2 -10355.881} C_VEL
LIN {X 0,Y 411.483,Z 494.043,A -85,B 0,C 180,E1 -10357.853,E2 -10357.853} C_VEL
LIN {X 0,Y 411.284,Z 494.067,A -85,B 0,C 180,E1 -10361.832,E2 -10361.832} C_VEL
LIN {X 0,Y 411.262,Z 494.068,A -85,B 0,C 180,E1 -10364.852,E2 -10364.852} C_VEL
LIN {X 0,Y 411.253,Z 494.071,A -85,B 0,C 180,E1 -10367.914,E2 -10367.914} C_VEL
LIN {X 0,Y 411.197,Z 494.075,A -85,B 0,C 180,E1 -10371.033,E2 -10371.033} C_VEL
LIN {X 0,Y 411.227,Z 494.076,A -85,B 0,C 180,E1 -10374.215,E2 -10374.215} C_VEL
LIN {X 0,Y 411.259,Z 494.068,A -85,B 0,C 180,E1 -10377.477,E2 -10377.477} C_VEL
LIN {X 0,Y 411.198,Z 494.077,A -85,B 0,C 180,E1 -10380.846,E2 -10380.846} C_VEL
LIN {X 0,Y 411.206,Z 494.078,A -85,B 0,C 180,E1 -10384.333,E2 -10384.333} C_VEL
LIN {X 0,Y 411.2,Z 494.079,A -85,B 0,C 180,E1 -10387.972,E2 -10387.972} C_VEL
LIN {X 0,Y 411.182,Z 494.08,A -85,B 0,C 180,E1 -10390.503,E2 -10390.503} C_VEL
LIN {X 0,Y 411.176,Z 494.079,A -85,B 0,C 180,E1 -10393.132,E2 -10393.132} C_VEL
LIN {X 0,Y 411.235,Z 494.075,A -85,B 0,C 180,E1 -10395.871,E2 -10395.871} C_VEL
LIN {X 0,Y 411.208,Z 494.075,A -85,B 0,C 180,E1 -10398.764,E2 -10398.764} C_VEL
LIN {X 0,Y 411.202,Z 494.079,A -85,B 0,C 180,E1 -10402.027,E2 -10402.027} C_VEL
LIN {X 0,Y 411.203,Z 494.078,A -85,B 0,C 180,E1 -10405.666,E2 -10405.666} C_VEL
LIN {X 0,Y 411.187,Z 494.077,A -85,B 0,C 180,E1 -10409.152,E2 -10409.152} C_VEL
LIN {X 0,Y 411.256,Z 494.07,A -85,B 0,C 180,E1 -10412.522,E2 -10412.522} C_VEL
LIN {X 0,Y 411.225,Z 494.076,A -85,B 0,C 180,E1 -10415.784,E2 -10415.784} C_VEL
LIN {X 0,Y 411.194,Z 494.077,A -85,B 0,C 180,E1 -10418.966,E2 -10418.966} C_VEL
LIN {X 0,Y 411.25,Z 494.073,A -85,B 0,C 180,E1 -10422.085,E2 -10422.085} C_VEL
LIN {X 0,Y 411.26,Z 494.069,A -85,B 0,C 180,E1 -10425.147,E2 -10425.147} C_VEL
LIN {X 0,Y 411.296,Z 494.067,A -85,B 0,C 180,E1 -10428.168,E2 -10428.168} C_VEL
LIN {X 0,Y 411.479,Z 494.043,A -85,B 0,C 180,E1 -10432.147,E2 -10432.147} C_VEL
LIN {X 0,Y 411.473,Z 494.045,A -85,B 0,C 180,E1 -10434.118,E2 -10434.118} C_VEL
LIN {X 0,Y 411.512,Z 494.04,A -85,B 0,C 180,E1 -10438.042,E2 -10438.042} C_VEL
LIN {X 0,Y 411.64,Z 494.025,A -85,B 0,C 180,E1 -10440,E2 -10440} C_VEL
LIN {X 0,Y 411.465,Z 494.043,A -85,B 0,C 180,E1 -10442.937,E2 -10442.937} C_VEL
LIN {X 0,Y 411.458,Z 494.043,A -85,B 0,C 180,E1 -10446.867,E2 -10446.867} C_VEL
LIN {X 0,Y 411.302,Z 494.066,A -85,B 0,C 180,E1 -10449.838,E2 -10449.838} C_VEL
LIN {X 0,Y 411.302,Z 494.063,A -85,B 0,C 180,E1 -10453.104,E2 -10453.104} C_VEL
LIN {X 0,Y 411.26,Z 494.069,A -85,B 0,C 180,E1 -10456.869,E2 -10456.869} C_VEL
LIN {X 0,Y 411.227,Z 494.076,A -85,B 0,C 180,E1 -10459.987,E2 -10459.987} C_VEL
LIN {X 0,Y 411.2,Z 494.078,A -85,B 0,C 180,E1 -10463.148,E2 -10463.148} C_VEL
LIN {X 0,Y 411.235,Z 494.072,A -85,B 0,C 180,E1 -10466.381,E2 -10466.381} C_VEL
LIN {X 0,Y 411.209,Z 494.079,A -85,B 0,C 180,E1 -10469.712,E2 -10469.712} C_VEL
LIN {X 0,Y 411.204,Z 494.077,A -85,B 0,C 180,E1 -10473.156,E2 -10473.156} C_VEL
LIN {X 0,Y 411.193,Z 494.076,A -85,B 0,C 180,E1 -10476.553,E2 -10476.553} C_VEL
LIN {X 0,Y 411.213,Z 494.077,A -85,B 0,C 180,E1 -10479.729,E2 -10479.729} C_VEL
LIN {X 0,Y 411.175,Z 494.082,A -85,B 0,C 180,E1 -10483.133,E2 -10483.133} C_VEL
LIN {X 0,Y 411.166,Z 494.083,A -85,B 0,C 180,E1 -10485.881,E2 -10485.881} C_VEL
LIN {X 0,Y 411.198,Z 494.077,A -85,B 0,C 180,E1 -10488.766,E2 -10488.766} C_VEL
LIN {X 0,Y 411.203,Z 494.078,A -85,B 0,C 180,E1 -10492.028,E2 -10492.028} C_VEL
LIN {X 0,Y 411.223,Z 494.182,A -85,B 0,C 180,E1 -10493.946,E2 -10493.946} C_VEL
LIN {X 0,Y 412.289,Z 499.997,A -85,B 0,C 180,E1 -10496.644,E2 -10496.644} C_VEL
LIN {X 0,Y 412.763,Z 503.827,A -85,B 0,C 180,E1 -10498.357,E2 -10498.357} C_VEL
LIN {X 0,Y 412.266,Z 511.211,A -85,B 0,C 180,E1 -10501.49,E2 -10501.49} C_VEL
LIN {X 0,Y 411.661,Z 519.223,A -85,B 0,C 180,E1 -10504.8,E2 -10504.8} C_VEL
LIN {X 0,Y 411.203,Z 526.906,A -85,B 0,C 180,E1 -10507.914,E2 -10507.914} C_VEL
LIN {X 0,Y 410.719,Z 536.042,A -85,B 0,C 180,E1 -10511.545,E2 -10511.545} C_VEL
LIN {X 0,Y 410.425,Z 543.843,A -85,B 0,C 180,E1 -10514.609,E2 -10514.609} C_VEL
LIN {X 0,Y 410.278,Z 548.631,A -85,B 0,C 180,E1 -10516.47,E2 -10516.47} C_VEL
LIN {X 0,Y 411.722,Z 562.786,A -85,B 0,C 180,E1 -10517.048,E2 -10517.048} C_VEL
LIN {X 0,Y 412.394,Z 571.918,A -85,B 0,C 180,E1 -10517.576,E2 -10517.576} C_VEL
LIN {X 0,Y 412.063,Z 580.567,A -85,B 0,C 180,E1 -10518.19,E2 -10518.19} C_VEL
LIN {X 0,Y 411.648,Z 588.818,A -85,B 0,C 180,E1 -10518.927,E2 -10518.927} C_VEL
LIN {X 0,Y 411.243,Z 596.62,A -85,B 0,C 180,E1 -10519.788,E2 -10519.788} C_VEL
LIN {X 0,Y 410.925,Z 603.046,A -85,B 0,C 180,E1 -10520.65,E2 -10520.65} C_VEL
LIN {X 0,Y 410.533,Z 610.561,A -85,B 0,C 180,E1 -10521.881,E2 -10521.881} C_VEL
LIN {X 0,Y 410.273,Z 616.445,A -85,B 0,C 180,E1 -10523.114,E2 -10523.114} C_VEL
LIN {X 0,Y 410.104,Z 620.249,A -85,B 0,C 180,E1 -10524.099,E2 -10524.099} C_VEL
LIN {X 0,Y 410.033,Z 624.583,A -85,B 0,C 180,E1 -10525.577,E2 -10525.577} C_VEL
LIN {X 0,Y 410.002,Z 627.59,A -85,B 0,C 180,E1 -10527.053,E2 -10527.053} C_VEL
LIN {X 0,Y 410.021,Z 628.92,A -85,B 0,C 180,E1 -10528.036,E2 -10528.036} C_VEL
LIN {X 0,Y 409.976,Z 629.749,A -85,B 0,C 180,E1 -10529.018,E2 -10529.018} C_VEL
LIN {X 0,Y 409.978,Z 630.049,A -85,B 0,C 180,E1 -10530,E2 -10530} C_VEL
LIN {X 0,Y 409.976,Z 629.761,A -85,B 0,C 180,E1 -10530.983,E2 -10530.983} C_VEL
LIN {X 0,Y 410.02,Z 628.98,A -85,B 0,C 180,E1 -10531.965,E2 -10531.965} C_VEL
LIN {X 0,Y 409.987,Z 627.701,A -85,B 0,C 180,E1 -10532.948,E2 -10532.948} C_VEL
LIN {X 0,Y 410.034,Z 624.742,A -85,B 0,C 180,E1 -10534.424,E2 -10534.424} C_VEL
LIN {X 0,Y 410.118,Z 622.024,A -85,B 0,C 180,E1 -10535.409,E2 -10535.409} C_VEL
LIN {X 0,Y 410.277,Z 616.782,A -85,B 0,C 180,E1 -10536.887,E2 -10536.887} C_VEL
LIN {X 0,Y 410.606,Z 609.897,A -85,B 0,C 180,E1 -10538.366,E2 -10538.366} C_VEL
LIN {X 0,Y 411.061,Z 602.562,A -85,B 0,C 180,E1 -10539.596,E2 -10539.596} C_VEL
LIN {X 0,Y 411.517,Z 595.36,A -85,B 0,C 180,E1 -10540.579,E2 -10540.579} C_VEL
LIN {X 0,Y 412.043,Z 586.594,A -85,B 0,C 180,E1 -10541.562,E2 -10541.562} C_VEL
LIN {X 0,Y 412.7,Z 577.18,A -85,B 0,C 180,E1 -10542.416,E2 -10542.416} C_VEL
LIN {X 0,Y 412.653,Z 569.533,A -85,B 0,C 180,E1 -10542.994,E2 -10542.994} C_VEL
LIN {X 0,Y 411.826,Z 557.321,A -85,B 0,C 180,E1 -10543.749,E2 -10543.749} C_VEL
LIN {X 0,Y 410.229,Z 546.872,A -85,B 0,C 180,E1 -10544.257,E2 -10544.257} C_VEL
LIN {X 0,Y 410.526,Z 539.216,A -85,B 0,C 180,E1 -10547.434,E2 -10547.434} C_VEL
LIN {X 0,Y 410.859,Z 532.013,A -85,B 0,C 180,E1 -10550.529,E2 -10550.529} C_VEL
LIN {X 0,Y 411.333,Z 523.897,A -85,B 0,C 180,E1 -10554.209,E2 -10554.209} C_VEL
LIN {X 0,Y 411.898,Z 517.278,A -85,B 0,C 180,E1 -10557.432,E2 -10557.432} C_VEL
LIN {X 0,Y 412.646,Z 511.096,A -85,B 0,C 180,E1 -10560.727,E2 -10560.727} C_VEL
LIN {X 0,Y 413.072,Z 506.494,A -85,B 0,C 180,E1 -10563.521,E2 -10563.521} C_VEL
LIN {X 0,Y 412.892,Z 503.913,A -85,B 0,C 180,E1 -10565.362,E2 -10565.362} C_VEL
LIN {X 0,Y 412.338,Z 500.439,A -85,B 0,C 180,E1 -10568.369,E2 -10568.369} C_VEL
LIN {X 0,Y 411.88,Z 497.873,A -85,B 0,C 180,E1 -10571.342,E2 -10571.342} C_VEL
LIN {X 0,Y 411.545,Z 496.147,A -85,B 0,C 180,E1 -10574.441,E2 -10574.441} C_VEL
LIN {X 0,Y 411.415,Z 495.372,A -85,B 0,C 180,E1 -10577.27,E2 -10577.27} C_VEL
LIN {X 0,Y 411.416,Z 495.343,A -85,B 0,C 180,E1 -10580.239,E2 -10580.239} C_VEL
LIN {X 0,Y 411.501,Z 496.049,A -85,B 0,C 180,E1 -10583.39,E2 -10583.39} C_VEL
LIN {X 0,Y 411.682,Z 497.525,A -85,B 0,C 180,E1 -10586.773,E2 -10586.773} C_VEL
LIN {X 0,Y 411.556,Z 498.988,A -85,B 0,C 180,E1 -10589.183,E2 -10589.183} C_VEL
LIN {X 0,Y 411.206,Z 501.584,A -85,B 0,C 180,E1 -10592.716,E2 -10592.716} C_VEL
LIN {X 0,Y 410.922,Z 504.142,A -85,B 0,C 180,E1 -10595.766,E2 -10595.766} C_VEL
LIN {X 0,Y 410.762,Z 507.036,A -85,B 0,C 180,E1 -10598.943,E2 -10598.943} C_VEL
LIN {X 0,Y 410.584,Z 510.084,A -85,B 0,C 180,E1 -10602.055,E2 -10602.055} C_VEL
LIN {X 0,Y 410.455,Z 513.251,A -85,B 0,C 180,E1 -10605.118,E2 -10605.118} C_VEL
LIN {X 0,Y 410.461,Z 514.231,A -85,B 0,C 180,E1 -10605.894,E2 -10605.894} C_VEL
LIN {X 0,Y 413.089,Z 524.853,A -85,B 0,C 180,E1 -10606.538,E2 -10606.538} C_VEL
LIN {X 0,Y 413.935,Z 530.53,A -85,B 0,C 180,E1 -10606.918,E2 -10606.918} C_VEL
LIN {X 0,Y 413.363,Z 541.422,A -85,B 0,C 180,E1 -10607.73,E2 -10607.73} C_VEL
LIN {X 0,Y 412.77,Z 550.435,A -85,B 0,C 180,E1 -10608.584,E2 -10608.584} C_VEL
LIN {X 0,Y 412.316,Z 557.793,A -85,B 0,C 180,E1 -10609.442,E2 -10609.442} C_VEL
LIN {X 0,Y 411.731,Z 566.377,A -85,B 0,C 180,E1 -10610.668,E2 -10610.668} C_VEL
LIN {X 0,Y 411.229,Z 573.082,A -85,B 0,C 180,E1 -10611.895,E2 -10611.895} C_VEL
LIN {X 0,Y 410.939,Z 578.455,A -85,B 0,C 180,E1 -10613.124,E2 -10613.124} C_VEL
LIN {X 0,Y 410.523,Z 581.974,A -85,B 0,C 180,E1 -10614.104,E2 -10614.104} C_VEL
LIN {X 0,Y 410.466,Z 585.953,A -85,B 0,C 180,E1 -10615.581,E2 -10615.581} C_VEL
LIN {X 0,Y 410.39,Z 587.07,A -85,B 0,C 180,E1 -10616.072,E2 -10616.072} C_VEL
LIN {X 0,Y 410.207,Z 588.691,A -85,B 0,C 180,E1 -10617.054,E2 -10617.054} C_VEL
LIN {X 0,Y 410.104,Z 589.789,A -85,B 0,C 180,E1 -10618.036,E2 -10618.036} C_VEL
LIN {X 0,Y 410.008,Z 590.401,A -85,B 0,C 180,E1 -10619.018,E2 -10619.018} C_VEL
LIN {X 0,Y 409.981,Z 590.532,A -85,B 0,C 180,E1 -10620,E2 -10620} C_VEL
LIN {X 0,Y 409.994,Z 590.129,A -85,B 0,C 180,E1 -10620.982,E2 -10620.982} C_VEL
LIN {X 0,Y 410.073,Z 589.134,A -85,B 0,C 180,E1 -10621.964,E2 -10621.964} C_VEL
LIN {X 0,Y 410.181,Z 586.767,A -85,B 0,C 180,E1 -10623.438,E2 -10623.438} C_VEL
LIN {X 0,Y 410.262,Z 583.031,A -85,B 0,C 180,E1 -10624.914,E2 -10624.914} C_VEL
LIN {X 0,Y 410.428,Z 579.821,A -85,B 0,C 180,E1 -10625.897,E2 -10625.897} C_VEL
LIN {X 0,Y 410.728,Z 575.11,A -85,B 0,C 180,E1 -10627.045,E2 -10627.045} C_VEL
LIN {X 0,Y 410.877,Z 569.749,A -85,B 0,C 180,E1 -10628.112,E2 -10628.112} C_VEL
LIN {X 0,Y 411.205,Z 563.769,A -85,B 0,C 180,E1 -10629.096,E2 -10629.096} C_VEL
LIN {X 0,Y 411.638,Z 556.53,A -85,B 0,C 180,E1 -10630.079,E2 -10630.079} C_VEL
LIN {X 0,Y 412.016,Z 548.869,A -85,B 0,C 180,E1 -10630.939,E2 -10630.939} C_VEL
LIN {X 0,Y 412.385,Z 540.907,A -85,B 0,C 180,E1 -10631.676,E2 -10631.676} C_VEL
LIN {X 0,Y 412.839,Z 530.998,A -85,B 0,C 180,E1 -10632.411,E2 -10632.411} C_VEL
LIN {X 0,Y 412.712,Z 526.948,A -85,B 0,C 180,E1 -10632.665,E2 -10632.665} C_VEL
LIN {X 0,Y 411.043,Z 516.682,A -85,B 0,C 180,E1 -10633.224,E2 -10633.224} C_VEL
LIN {X 0,Y 410.192,Z 511.474,A -85,B 0,C 180,E1 -10633.462,E2 -10633.462} C_VEL
LIN {X 0,Y 410.177,Z 506.824,A -85,B 0,C 180,E1 -10636.935,E2 -10636.935} C_VEL
LIN {X 0,Y 410.256,Z 502.737,A -85,B 0,C 180,E1 -10640.036,E2 -10640.036} C_VEL
LIN {X 0,Y 410.364,Z 498.662,A -85,B 0,C 180,E1 -10643.198,E2 -10643.198} C_VEL
LIN {X 0,Y 410.615,Z 494.451,A -85,B 0,C 180,E1 -10646.593,E2 -10646.593} C_VEL
LIN {X 0,Y 410.957,Z 497.624,A -85,B 0,C 180,E1 -10648.053,E2 -10648.053} C_VEL
LIN {X 0,Y 410.812,Z 504.408,A -85,B 0,C 180,E1 -10651.198,E2 -10651.198} C_VEL
LIN {X 0,Y 410.745,Z 509.961,A -85,B 0,C 180,E1 -10653.786,E2 -10653.786} C_VEL
LIN {X 0,Y 410.573,Z 516.4,A -85,B 0,C 180,E1 -10656.807,E2 -10656.807} C_VEL
LIN {X 0,Y 410.407,Z 523.281,A -85,B 0,C 180,E1 -10660.057,E2 -10660.057} C_VEL
LIN {X 0,Y 410.384,Z 527.71,A -85,B 0,C 180,E1 -10662.164,E2 -10662.164} C_VEL
LIN {X 0,Y 412.681,Z 541.37,A -85,B 0,C 180,E1 -10662.802,E2 -10662.802} C_VEL
LIN {X 0,Y 413.336,Z 547.75,A -85,B 0,C 180,E1 -10663.186,E2 -10663.186} C_VEL
LIN {X 0,Y 412.751,Z 559.112,A -85,B 0,C 180,E1 -10663.995,E2 -10663.995} C_VEL
LIN {X 0,Y 412.293,Z 567.756,A -85,B 0,C 180,E1 -10664.802,E2 -10664.802} C_VEL
LIN {X 0,Y 411.841,Z 574.767,A -85,B 0,C 180,E1 -10665.6,E2 -10665.6} C_VEL
LIN {X 0,Y 411.373,Z 581.715,A -85,B 0,C 180,E1 -10666.556,E2 -10666.556} C_VEL
LIN {X 0,Y 410.932,Z 588.685,A -85,B 0,C 180,E1 -10667.731,E2 -10667.731} C_VEL
LIN {X 0,Y 410.539,Z 595.149,A -85,B 0,C 180,E1 -10669.134,E2 -10669.134} C_VEL
LIN {X 0,Y 410.279,Z 599.722,A -85,B 0,C 180,E1 -10670.43,E2 -10670.43} C_VEL
LIN {X 0,Y 410.154,Z 602.199,A -85,B 0,C 180,E1 -10671.286,E2 -10671.286} C_VEL
LIN {X 0,Y 410.066,Z 603.906,A -85,B 0,C 180,E1 -10672.035,E2 -10672.035} C_VEL
LIN {X 0,Y 409.874,Z 606.667,A -85,B 0,C 180,E1 -10673.697,E2 -10673.697} C_VEL
LIN {X 0,Y 409.767,Z 607.914,A -85,B 0,C 180,E1 -10675.528,E2 -10675.528} C_VEL
LIN {X 0,Y 409.775,Z 607.653,A -85,B 0,C 180,E1 -10677.182,E2 -10677.182} C_VEL
LIN {X 0,Y 409.916,Z 605.496,A -85,B 0,C 180,E1 -10679.045,E2 -10679.045} C_VEL
LIN {X 0,Y 410.046,Z 603.263,A -85,B 0,C 180,E1 -10680.195,E2 -10680.195} C_VEL
LIN {X 0,Y 410.198,Z 600.279,A -85,B 0,C 180,E1 -10681.332,E2 -10681.332} C_VEL
LIN {X 0,Y 410.42,Z 596.473,A -85,B 0,C 180,E1 -10682.461,E2 -10682.461} C_VEL
LIN {X 0,Y 410.755,Z 590.465,A -85,B 0,C 180,E1 -10683.859,E2 -10683.859} C_VEL
LIN {X 0,Y 411.233,Z 582.461,A -85,B 0,C 180,E1 -10685.28,E2 -10685.28} C_VEL
LIN {X 0,Y 411.673,Z 574.778,A -85,B 0,C 180,E1 -10686.347,E2 -10686.347} C_VEL
LIN {X 0,Y 412.125,Z 567.497,A -85,B 0,C 180,E1 -10687.174,E2 -10687.174} C_VEL
LIN {X 0,Y 412.536,Z 558.715,A -85,B 0,C 180,E1 -10687.988,E2 -10687.988} C_VEL
LIN {X 0,Y 413.102,Z 547.049,A -85,B 0,C 180,E1 -10688.806,E2 -10688.806} C_VEL
LIN {X 0,Y 411.754,Z 537.191,A -85,B 0,C 180,E1 -10689.355,E2 -10689.355} C_VEL
LIN {X 0,Y 410.166,Z 527.795,A -85,B 0,C 180,E1 -10689.763,E2 -10689.763} C_VEL
LIN {X 0,Y 410.277,Z 521.305,A -85,B 0,C 180,E1 -10693.069,E2 -10693.069} C_VEL
LIN {X 0,Y 410.373,Z 515.304,A -85,B 0,C 180,E1 -10696.127,E2 -10696.127} C_VEL
LIN {X 0,Y 410.579,Z 511.387,A -85,B 0,C 180,E1 -10698.146,E2 -10698.146} C_VEL
LIN {X 0,Y 410.651,Z 505.482,A -85,B 0,C 180,E1 -10701.139,E2 -10701.139} C_VEL
LIN {X 0,Y 410.777,Z 499.597,A -85,B 0,C 180,E1 -10704.107,E2 -10704.107} C_VEL
LIN {X 0,Y 410.896,Z 494.118,A -85,B 0,C 180,E1 -10706.936,E2 -10706.936} C_VEL
LIN {X 0,Y 411.633,Z 494.024,A -85,B 0,C 180,E1 -10710,E2 -10710} C_VEL
LIN {X 0,Y 411.493,Z 494.04,A -85,B 0,C 180,E1 -10711.735,E2 -10711.735} C_VEL
LIN {X 0,Y 410.883,Z 494.121,A -85,B 0,C 180,E1 -10712.55,E2 -10712.55} C_VEL
LIN {X 0,Y 408.049,Z 494.479,A -85,B 0,C 180,E1 -10713.874,E2 -10713.874} C_VEL
LIN {X 0,Y 405.599,Z 494.782,A -85,B 0,C 180,E1 -10714.943,E2 -10714.943} C_VEL
LIN {X 0,Y 404.521,Z 494.912,A -85,B 0,C 180,E1 -10715.769,E2 -10715.769} C_VEL
LIN {X 0,Y 404.422,Z 494.922,A -85,B 0,C 180,E1 -10716.05,E2 -10716.05} C_VEL
LIN {X 0,Y 404.424,Z 494.923,A -85,B 0,C 180,E1 -10717.991,E2 -10717.991} C_VEL
LIN {X 0,Y 404.257,Z 494.943,A -85,B 0,C 180,E1 -10722.041,E2 -10722.041} C_VEL
LIN {X 0,Y 404.208,Z 494.946,A -85,B 0,C 180,E1 -10725.117,E2 -10725.117} C_VEL
LIN {X 0,Y 404.211,Z 494.951,A -85,B 0,C 180,E1 -10728.237,E2 -10728.237} C_VEL
LIN {X 0,Y 404.139,Z 494.954,A -85,B 0,C 180,E1 -10731.419,E2 -10731.419} C_VEL
LIN {X 0,Y 404.177,Z 494.952,A -85,B 0,C 180,E1 -10734.665,E2 -10734.665} C_VEL
LIN {X 0,Y 404.198,Z 494.952,A -85,B 0,C 180,E1 -10737.999,E2 -10737.999} C_VEL
LIN {X 0,Y 404.142,Z 494.956,A -85,B 0,C 180,E1 -10741.558,E2 -10741.558} C_VEL
LIN {X 0,Y 404.185,Z 494.949,A -85,B 0,C 180,E1 -10745.015,E2 -10745.015} C_VEL
LIN {X 0,Y 404.158,Z 494.953,A -85,B 0,C 180,E1 -10748.756,E2 -10748.756} C_VEL
LIN {X 0,Y 404.123,Z 494.958,A -85,B 0,C 180,E1 -10751.6,E2 -10751.6} C_VEL
LIN {X 0,Y 404.155,Z 494.955,A -85,B 0,C 180,E1 -10754.523,E2 -10754.523} C_VEL
LIN {X 0,Y 404.209,Z 494.946,A -85,B 0,C 180,E1 -10757.305,E2 -10757.305} C_VEL
LIN {X 0,Y 404.167,Z 494.955,A -85,B 0,C 180,E1 -10759.955,E2 -10759.955} C_VEL
LIN {X 0,Y 404.138,Z 494.955,A -85,B 0,C 180,E1 -10763.124,E2 -10763.124} C_VEL
LIN {X 0,Y 404.142,Z 494.958,A -85,B 0,C 180,E1 -10766.187,E2 -10766.187} C_VEL
LIN {X 0,Y 404.143,Z 494.958,A -85,B 0,C 180,E1 -10769.715,E2 -10769.715} C_VEL
LIN {X 0,Y 404.193,Z 494.949,A -85,B 0,C 180,E1 -10773.123,E2 -10773.123} C_VEL
LIN {X 0,Y 404.175,Z 494.951,A -85,B 0,C 180,E1 -10775.334,E2 -10775.334} C_VEL
LIN {X 0,Y 404.136,Z 494.956,A -85,B 0,C 180,E1 -10778.58,E2 -10778.58} C_VEL
LIN {X 0,Y 404.208,Z 494.95,A -85,B 0,C 180,E1 -10781.762,E2 -10781.762} C_VEL
LIN {X 0,Y 404.205,Z 494.947,A -85,B 0,C 180,E1 -10784.882,E2 -10784.882} C_VEL
LIN {X 0,Y 404.267,Z 494.942,A -85,B 0,C 180,E1 -10787.959,E2 -10787.959} C_VEL
LIN {X 0,Y 404.431,Z 494.921,A -85,B 0,C 180,E1 -10792.099,E2 -10792.099} C_VEL
LIN {X 0,Y 404.421,Z 494.923,A -85,B 0,C 180,E1 -10794.015,E2 -10794.015} C_VEL
LIN {X 0,Y 404.481,Z 494.916,A -85,B 0,C 180,E1 -10798.008,E2 -10798.008} C_VEL
LIN {X 0,Y 404.609,Z 494.9,A -85,B 0,C 180,E1 -10800,E2 -10800} C_VEL
LIN {X 0,Y 404.422,Z 494.92,A -85,B 0,C 180,E1 -10802.988,E2 -10802.988} C_VEL
LIN {X 0,Y 404.409,Z 494.921,A -85,B 0,C 180,E1 -10806.987,E2 -10806.987} C_VEL
LIN {X 0,Y 404.264,Z 494.942,A -85,B 0,C 180,E1 -10810.011,E2 -10810.011} C_VEL
LIN {X 0,Y 404.263,Z 494.941,A -85,B 0,C 180,E1 -10813.211,E2 -10813.211} C_VEL
LIN {X 0,Y 404.213,Z 494.947,A -85,B 0,C 180,E1 -10817.007,E2 -10817.007} C_VEL
LIN {X 0,Y 404.161,Z 494.953,A -85,B 0,C 180,E1 -10820.352,E2 -10820.352} C_VEL
LIN {X 0,Y 404.166,Z 494.955,A -85,B 0,C 180,E1 -10823.575,E2 -10823.575} C_VEL
LIN {X 0,Y 404.181,Z 494.953,A -85,B 0,C 180,E1 -10825.767,E2 -10825.767} C_VEL
LIN {X 0,Y 404.195,Z 494.95,A -85,B 0,C 180,E1 -10828,E2 -10828} C_VEL
LIN {X 0,Y 404.143,Z 494.958,A -85,B 0,C 180,E1 -10831.56,E2 -10831.56} C_VEL
LIN {X 0,Y 404.183,Z 494.951,A -85,B 0,C 180,E1 -10835.016,E2 -10835.016} C_VEL
LIN {X 0,Y 404.155,Z 494.953,A -85,B 0,C 180,E1 -10838.757,E2 -10838.757} C_VEL
LIN {X 0,Y 404.122,Z 494.961,A -85,B 0,C 180,E1 -10841.6,E2 -10841.6} C_VEL
LIN {X 0,Y 404.146,Z 494.954,A -85,B 0,C 180,E1 -10844.523,E2 -10844.523} C_VEL
LIN {X 0,Y 404.168,Z 494.954,A -85,B 0,C 180,E1 -10847.301,E2 -10847.301} C_VEL
LIN {X 0,Y 404.166,Z 494.953,A -85,B 0,C 180,E1 -10849.956,E2 -10849.956} C_VEL
LIN {X 0,Y 404.171,Z 494.955,A -85,B 0,C 180,E1 -10853.6,E2 -10853.6} C_VEL
LIN {X 0,Y 404.186,Z 495.009,A -85,B 0,C 180,E1 -10853.759,E2 -10853.759} C_VEL
LIN {X 0,Y 405.186,Z 500.513,A -85,B 0,C 180,E1 -10856.363,E2 -10856.363} C_VEL
LIN {X 0,Y 405.76,Z 504.237,A -85,B 0,C 180,E1 -10858.071,E2 -10858.071} C_VEL
LIN {X 0,Y 405.325,Z 510.886,A -85,B 0,C 180,E1 -10860.956,E2 -10860.956} C_VEL
LIN {X 0,Y 404.641,Z 519.464,A -85,B 0,C 180,E1 -10864.577,E2 -10864.577} C_VEL
LIN {X 0,Y 404.107,Z 527.851,A -85,B 0,C 180,E1 -10868.043,E2 -10868.043} C_VEL
LIN {X 0,Y 403.615,Z 536.962,A -85,B 0,C 180,E1 -10871.735,E2 -10871.735} C_VEL
LIN {X 0,Y 403.316,Z 544.732,A -85,B 0,C 180,E1 -10874.848,E2 -10874.848} C_VEL
LIN {X 0,Y 403.203,Z 548.3,A -85,B 0,C 180,E1 -10876.265,E2 -10876.265} C_VEL
LIN {X 0,Y 404.436,Z 560.167,A -85,B 0,C 180,E1 -10876.715,E2 -10876.715} C_VEL
LIN {X 0,Y 405.379,Z 571.506,A -85,B 0,C 180,E1 -10877.357,E2 -10877.357} C_VEL
LIN {X 0,Y 405.108,Z 580.199,A -85,B 0,C 180,E1 -10877.985,E2 -10877.985} C_VEL
LIN {X 0,Y 404.665,Z 588.48,A -85,B 0,C 180,E1 -10878.733,E2 -10878.733} C_VEL
LIN {X 0,Y 404.236,Z 596.306,A -85,B 0,C 180,E1 -10879.609,E2 -10879.609} C_VEL
LIN {X 0,Y 403.872,Z 602.75,A -85,B 0,C 180,E1 -10880.485,E2 -10880.485} C_VEL
LIN {X 0,Y 403.544,Z 608.866,A -85,B 0,C 180,E1 -10881.488,E2 -10881.488} C_VEL
LIN {X 0,Y 403.282,Z 615.1,A -85,B 0,C 180,E1 -10882.742,E2 -10882.742} C_VEL
LIN {X 0,Y 403.016,Z 620.005,A -85,B 0,C 180,E1 -10883.995,E2 -10883.995} C_VEL
LIN {X 0,Y 402.963,Z 624.358,A -85,B 0,C 180,E1 -10885.499,E2 -10885.499} C_VEL
LIN {X 0,Y 402.9,Z 627.374,A -85,B 0,C 180,E1 -10887.001,E2 -10887.001} C_VEL
LIN {X 0,Y 402.933,Z 628.714,A -85,B 0,C 180,E1 -10888.001,E2 -10888.001} C_VEL
LIN {X 0,Y 402.901,Z 629.553,A -85,B 0,C 180,E1 -10889.001,E2 -10889.001} C_VEL
LIN {X 0,Y 402.9,Z 629.856,A -85,B 0,C 180,E1 -10890.001,E2 -10890.001} C_VEL
LIN {X 0,Y 402.901,Z 629.575,A -85,B 0,C 180,E1 -10891,E2 -10891} C_VEL
LIN {X 0,Y 402.931,Z 628.802,A -85,B 0,C 180,E1 -10892,E2 -10892} C_VEL
LIN {X 0,Y 402.885,Z 627.532,A -85,B 0,C 180,E1 -10893,E2 -10893} C_VEL
LIN {X 0,Y 402.964,Z 624.582,A -85,B 0,C 180,E1 -10894.502,E2 -10894.502} C_VEL
LIN {X 0,Y 403.017,Z 621.873,A -85,B 0,C 180,E1 -10895.504,E2 -10895.504} C_VEL
LIN {X 0,Y 403.21,Z 616.624,A -85,B 0,C 180,E1 -10897.009,E2 -10897.009} C_VEL
LIN {X 0,Y 403.581,Z 609.791,A -85,B 0,C 180,E1 -10898.513,E2 -10898.513} C_VEL
LIN {X 0,Y 404.043,Z 602.614,A -85,B 0,C 180,E1 -10899.765,E2 -10899.765} C_VEL
LIN {X 0,Y 404.616,Z 594.53,A -85,B 0,C 180,E1 -10900.889,E2 -10900.889} C_VEL
LIN {X 0,Y 405.102,Z 586.931,A -85,B 0,C 180,E1 -10901.763,E2 -10901.763} C_VEL
LIN {X 0,Y 405.789,Z 577.67,A -85,B 0,C 180,E1 -10902.631,E2 -10902.631} C_VEL
LIN {X 0,Y 405.846,Z 571.594,A -85,B 0,C 180,E1 -10903.115,E2 -10903.115} C_VEL
LIN {X 0,Y 405.387,Z 562.293,A -85,B 0,C 180,E1 -10903.753,E2 -10903.753} C_VEL
LIN {X 0,Y 403.911,Z 550.675,A -85,B 0,C 180,E1 -10904.421,E2 -10904.421} C_VEL
LIN {X 0,Y 403.188,Z 546.404,A -85,B 0,C 180,E1 -10904.641,E2 -10904.641} C_VEL
LIN {X 0,Y 403.479,Z 539.103,A -85,B 0,C 180,E1 -10907.748,E2 -10907.748} C_VEL
LIN {X 0,Y 403.813,Z 531.973,A -85,B 0,C 180,E1 -10910.903,E2 -10910.903} C_VEL
LIN {X 0,Y 404.377,Z 523.945,A -85,B 0,C 180,E1 -10914.653,E2 -10914.653} C_VEL
LIN {X 0,Y 405.011,Z 517.445,A -85,B 0,C 180,E1 -10917.939,E2 -10917.939} C_VEL
LIN {X 0,Y 405.783,Z 511.419,A -85,B 0,C 180,E1 -10921.305,E2 -10921.305} C_VEL
LIN {X 0,Y 406.103,Z 507.46,A -85,B 0,C 180,E1 -10923.831,E2 -10923.831} C_VEL
LIN {X 0,Y 405.829,Z 504.506,A -85,B 0,C 180,E1 -10926.072,E2 -10926.072} C_VEL
LIN {X 0,Y 405.339,Z 501.647,A -85,B 0,C 180,E1 -10928.718,E2 -10928.718} C_VEL
LIN {X 0,Y 404.919,Z 499.207,A -85,B 0,C 180,E1 -10931.726,E2 -10931.726} C_VEL
LIN {X 0,Y 404.618,Z 497.694,A -85,B 0,C 180,E1 -10934.59,E2 -10934.59} C_VEL
LIN {X 0,Y 404.512,Z 496.938,A -85,B 0,C 180,E1 -10937.345,E2 -10937.345} C_VEL
LIN {X 0,Y 404.475,Z 496.838,A -85,B 0,C 180,E1 -10939.992,E2 -10939.992} C_VEL
LIN {X 0,Y 404.528,Z 497.395,A -85,B 0,C 180,E1 -10943.052,E2 -10943.052} C_VEL
LIN {X 0,Y 404.699,Z 498.716,A -85,B 0,C 180,E1 -10946.468,E2 -10946.468} C_VEL
LIN {X 0,Y 404.622,Z 499.889,A -85,B 0,C 180,E1 -10948.595,E2 -10948.595} C_VEL
LIN {X 0,Y 404.267,Z 502.218,A -85,B 0,C 180,E1 -10952.006,E2 -10952.006} C_VEL
LIN {X 0,Y 403.939,Z 504.852,A -85,B 0,C 180,E1 -10955.319,E2 -10955.319} C_VEL
LIN {X 0,Y 403.748,Z 507.688,A -85,B 0,C 180,E1 -10958.559,E2 -10958.559} C_VEL
LIN {X 0,Y 403.548,Z 510.697,A -85,B 0,C 180,E1 -10961.731,E2 -10961.731} C_VEL
LIN {X 0,Y 403.412,Z 513.834,A -85,B 0,C 180,E1 -10964.852,E2 -10964.852} C_VEL
LIN {X 0,Y 403.424,Z 514.722,A -85,B 0,C 180,E1 -10965.53,E2 -10965.53} C_VEL
LIN {X 0,Y 406.383,Z 526.414,A -85,B 0,C 180,E1 -10966.293,E2 -10966.293} C_VEL
LIN {X 0,Y 407.135,Z 532.627,A -85,B 0,C 180,E1 -10966.735,E2 -10966.735} C_VEL
LIN {X 0,Y 406.525,Z 542.681,A -85,B 0,C 180,E1 -10967.52,E2 -10967.52} C_VEL
LIN {X 0,Y 405.995,Z 550.375,A -85,B 0,C 180,E1 -10968.264,E2 -10968.264} C_VEL
LIN {X 0,Y 405.416,Z 558.786,A -85,B 0,C 180,E1 -10969.26,E2 -10969.26} C_VEL
LIN {X 0,Y 404.787,Z 567.221,A -85,B 0,C 180,E1 -10970.506,E2 -10970.506} C_VEL
LIN {X 0,Y 404.259,Z 573.808,A -85,B 0,C 180,E1 -10971.754,E2 -10971.754} C_VEL
LIN {X 0,Y 403.93,Z 579.093,A -85,B 0,C 180,E1 -10973.004,E2 -10973.004} C_VEL
LIN {X 0,Y 403.497,Z 582.545,A -85,B 0,C 180,E1 -10974.001,E2 -10974.001} C_VEL
LIN {X 0,Y 403.424,Z 586.466,A -85,B 0,C 180,E1 -10975.504,E2 -10975.504} C_VEL
LIN {X 0,Y 403.151,Z 589.161,A -85,B 0,C 180,E1 -10977.002,E2 -10977.002} C_VEL
LIN {X 0,Y 403.033,Z 590.217,A -85,B 0,C 180,E1 -10978.001,E2 -10978.001} C_VEL
LIN {X 0,Y 402.932,Z 590.785,A -85,B 0,C 180,E1 -10979.001,E2 -10979.001} C_VEL
LIN {X 0,Y 402.903,Z 590.868,A -85,B 0,C 180,E1 -10980,E2 -10980} C_VEL
LIN {X 0,Y 402.919,Z 590.441,A -85,B 0,C 180,E1 -10981,E2 -10981} C_VEL
LIN {X 0,Y 403.005,Z 589.412,A -85,B 0,C 180,E1 -10981.999,E2 -10981.999} C_VEL
LIN {X 0,Y 403.103,Z 586.966,A -85,B 0,C 180,E1 -10983.499,E2 -10983.499} C_VEL
LIN {X 0,Y 403.198,Z 583.138,A -85,B 0,C 180,E1 -10985,E2 -10985} C_VEL
LIN {X 0,Y 403.451,Z 578.593,A -85,B 0,C 180,E1 -10986.324,E2 -10986.324} C_VEL
LIN {X 0,Y 403.717,Z 573.49,A -85,B 0,C 180,E1 -10987.502,E2 -10987.502} C_VEL
LIN {X 0,Y 403.918,Z 568.203,A -85,B 0,C 180,E1 -10988.505,E2 -10988.505} C_VEL
LIN {X 0,Y 404.29,Z 561.866,A -85,B 0,C 180,E1 -10989.506,E2 -10989.506} C_VEL
LIN {X 0,Y 404.797,Z 553.196,A -85,B 0,C 180,E1 -10990.63,E2 -10990.63} C_VEL
LIN {X 0,Y 405.29,Z 543.323,A -85,B 0,C 180,E1 -10991.63,E2 -10991.63} C_VEL
LIN {X 0,Y 405.751,Z 534.214,A -85,B 0,C 180,E1 -10992.356,E2 -10992.356} C_VEL
LIN {X 0,Y 405.7,Z 527.617,A -85,B 0,C 180,E1 -10992.799,E2 -10992.799} C_VEL
LIN {X 0,Y 404.08,Z 517.803,A -85,B 0,C 180,E1 -10993.35,E2 -10993.35} C_VEL
LIN {X 0,Y 403.099,Z 511.778,A -85,B 0,C 180,E1 -10993.633,E2 -10993.633} C_VEL
LIN {X 0,Y 403.146,Z 507.957,A -85,B 0,C 180,E1 -10996.501,E2 -10996.501} C_VEL
LIN {X 0,Y 403.213,Z 503.725,A -85,B 0,C 180,E1 -10999.741,E2 -10999.741} C_VEL
LIN {X 0,Y 403.302,Z 500.141,A -85,B 0,C 180,E1 -11002.543,E2 -11002.543} C_VEL
LIN {X 0,Y 403.418,Z 496.011,A -85,B 0,C 180,E1 -11005.819,E2 -11005.819} C_VEL
LIN {X 0,Y 403.537,Z 495.318,A -85,B 0,C 180,E1 -11006.506,E2 -11006.506} C_VEL
LIN {X 0,Y 403.927,Z 498.547,A -85,B 0,C 180,E1 -11008.02,E2 -11008.02} C_VEL
LIN {X 0,Y 403.746,Z 505.943,A -85,B 0,C 180,E1 -11011.481,E2 -11011.481} C_VEL
LIN {X 0,Y 403.621,Z 512.242,A -85,B 0,C 180,E1 -11014.465,E2 -11014.465} C_VEL
LIN {X 0,Y 403.509,Z 518.778,A -85,B 0,C 180,E1 -11017.561,E2 -11017.561} C_VEL
LIN {X 0,Y 403.304,Z 525.593,A -85,B 0,C 180,E1 -11020.804,E2 -11020.804} C_VEL
LIN {X 0,Y 403.321,Z 527.977,A -85,B 0,C 180,E1 -11021.925,E2 -11021.925} C_VEL
LIN {X 0,Y 405.155,Z 537.799,A -85,B 0,C 180,E1 -11022.361,E2 -11022.361} C_VEL
LIN {X 0,Y 406.424,Z 547.751,A -85,B 0,C 180,E1 -11022.937,E2 -11022.937} C_VEL
LIN {X 0,Y 405.9,Z 557.973,A -85,B 0,C 180,E1 -11023.654,E2 -11023.654} C_VEL
LIN {X 0,Y 405.393,Z 567.395,A -85,B 0,C 180,E1 -11024.532,E2 -11024.532} C_VEL
LIN {X 0,Y 404.848,Z 575.565,A -85,B 0,C 180,E1 -11025.48,E2 -11025.48} C_VEL
LIN {X 0,Y 404.336,Z 582.633,A -85,B 0,C 180,E1 -11026.486,E2 -11026.486} C_VEL
LIN {X 0,Y 403.817,Z 590.614,A -85,B 0,C 180,E1 -11027.921,E2 -11027.921} C_VEL
LIN {X 0,Y 403.43,Z 596.127,A -85,B 0,C 180,E1 -11029.211,E2 -11029.211} C_VEL
LIN {X 0,Y 403.269,Z 599.179,A -85,B 0,C 180,E1 -11030.069,E2 -11030.069} C_VEL
LIN {X 0,Y 403.088,Z 602.228,A -85,B 0,C 180,E1 -11031.121,E2 -11031.121} C_VEL
LIN {X 0,Y 402.914,Z 604.964,A -85,B 0,C 180,E1 -11032.374,E2 -11032.374} C_VEL
LIN {X 0,Y 402.809,Z 606.83,A -85,B 0,C 180,E1 -11033.614,E2 -11033.614} C_VEL
LIN {X 0,Y 402.695,Z 607.985,A -85,B 0,C 180,E1 -11035.111,E2 -11035.111} C_VEL
LIN {X 0,Y 402.664,Z 608.219,A -85,B 0,C 180,E1 -11036.046,E2 -11036.046} C_VEL
LIN {X 0,Y 402.702,Z 607.808,A -85,B 0,C 180,E1 -11037.247,E2 -11037.247} C_VEL
LIN {X 0,Y 402.795,Z 606.213,A -85,B 0,C 180,E1 -11038.755,E2 -11038.755} C_VEL
LIN {X 0,Y 402.964,Z 603.598,A -85,B 0,C 180,E1 -11040.189,E2 -11040.189} C_VEL
LIN {X 0,Y 403.107,Z 600.648,A -85,B 0,C 180,E1 -11041.35,E2 -11041.35} C_VEL
LIN {X 0,Y 403.382,Z 596.16,A -85,B 0,C 180,E1 -11042.693,E2 -11042.693} C_VEL
LIN {X 0,Y 403.693,Z 590.921,A -85,B 0,C 180,E1 -11043.922,E2 -11043.922} C_VEL
LIN {X 0,Y 404.19,Z 583.25,A -85,B 0,C 180,E1 -11045.335,E2 -11045.335} C_VEL
LIN {X 0,Y 404.647,Z 575.415,A -85,B 0,C 180,E1 -11046.454,E2 -11046.454} C_VEL
LIN {X 0,Y 405.157,Z 567.583,A -85,B 0,C 180,E1 -11047.363,E2 -11047.363} C_VEL
LIN {X 0,Y 405.553,Z 559.534,A -85,B 0,C 180,E1 -11048.124,E2 -11048.124} C_VEL
LIN {X 0,Y 406.101,Z 549.318,A -85,B 0,C 180,E1 -11048.888,E2 -11048.888} C_VEL
LIN {X 0,Y 405.735,Z 544.171,A -85,B 0,C 180,E1 -11049.2,E2 -11049.2} C_VEL
LIN {X 0,Y 404.048,Z 533.363,A -85,B 0,C 180,E1 -11049.769,E2 -11049.769} C_VEL
LIN {X 0,Y 403.104,Z 527.914,A -85,B 0,C 180,E1 -11049.999,E2 -11049.999} C_VEL
LIN {X 0,Y 403.23,Z 521.204,A -85,B 0,C 180,E1 -11053.458,E2 -11053.458} C_VEL
LIN {X 0,Y 403.434,Z 513.738,A -85,B 0,C 180,E1 -11057.303,E2 -11057.303} C_VEL
LIN {X 0,Y 403.546,Z 508.517,A -85,B 0,C 180,E1 -11059.97,E2 -11059.97} C_VEL
LIN {X 0,Y 403.701,Z 501.645,A -85,B 0,C 180,E1 -11063.502,E2 -11063.502} C_VEL
LIN {X 0,Y 403.858,Z 495.238,A -85,B 0,C 180,E1 -11066.757,E2 -11066.757} C_VEL
LIN {X 0,Y 403.849,Z 494.996,A -85,B 0,C 180,E1 -11067.007,E2 -11067.007} C_VEL
LIN {X 0,Y 404.601,Z 494.9,A -85,B 0,C 180,E1 -11069.999,E2 -11069.999} C_VEL
LIN {X 0,Y 404.424,Z 494.92,A -85,B 0,C 180,E1 -11072.988,E2 -11072.988} C_VEL
LIN {X 0,Y 404.422,Z 494.922,A -85,B 0,C 180,E1 -11076.05,E2 -11076.05} C_VEL
LIN {X 0,Y 403.714,Z 495.009,A -85,B 0,C 180,E1 -11076.88,E2 -11076.88} C_VEL
LIN {X 0,Y 400.811,Z 495.373,A -85,B 0,C 180,E1 -11078.229,E2 -11078.229} C_VEL
LIN {X 0,Y 398.361,Z 495.681,A -85,B 0,C 180,E1 -11079.319,E2 -11079.319} C_VEL
LIN {X 0,Y 397.296,Z 495.812,A -85,B 0,C 180,E1 -11080.162,E2 -11080.162} C_VEL
LIN {X 0,Y 397.201,Z 495.821,A -85,B 0,C 180,E1 -11080.447,E2 -11080.447} C_VEL
LIN {X 0,Y 397.227,Z 495.816,A -85,B 0,C 180,E1 -11083.32,E2 -11083.32} C_VEL
LIN {X 0,Y 397.182,Z 495.822,A -85,B 0,C 180,E1 -11087.155,E2 -11087.155} C_VEL
LIN {X 0,Y 397.103,Z 495.832,A -85,B 0,C 180,E1 -11090.729,E2 -11090.729} C_VEL
LIN {X 0,Y 397.133,Z 495.831,A -85,B 0,C 180,E1 -11094.018,E2 -11094.018} C_VEL
LIN {X 0,Y 397.194,Z 495.82,A -85,B 0,C 180,E1 -11097.389,E2 -11097.389} C_VEL
LIN {X 0,Y 397.084,Z 495.834,A -85,B 0,C 180,E1 -11100.881,E2 -11100.881} C_VEL
LIN {X 0,Y 397.125,Z 495.831,A -85,B 0,C 180,E1 -11104.493,E2 -11104.493} C_VEL
LIN {X 0,Y 397.106,Z 495.835,A -85,B 0,C 180,E1 -11108.274,E2 -11108.274} C_VEL
LIN {X 0,Y 397.088,Z 495.833,A -85,B 0,C 180,E1 -11110.908,E2 -11110.908} C_VEL
LIN {X 0,Y 397.103,Z 495.834,A -85,B 0,C 180,E1 -11113.647,E2 -11113.647} C_VEL
LIN {X 0,Y 397.163,Z 495.826,A -85,B 0,C 180,E1 -11116.511,E2 -11116.511} C_VEL
LIN {X 0,Y 397.122,Z 495.831,A -85,B 0,C 180,E1 -11119.55,E2 -11119.55} C_VEL
LIN {X 0,Y 397.096,Z 495.832,A -85,B 0,C 180,E1 -11122.79,E2 -11122.79} C_VEL
LIN {X 0,Y 397.116,Z 495.832,A -85,B 0,C 180,E1 -11126.282,E2 -11126.282} C_VEL
LIN {X 0,Y 397.103,Z 495.835,A -85,B 0,C 180,E1 -11130.135,E2 -11130.135} C_VEL
LIN {X 0,Y 397.192,Z 495.821,A -85,B 0,C 180,E1 -11132.61,E2 -11132.61} C_VEL
LIN {X 0,Y 397.131,Z 495.831,A -85,B 0,C 180,E1 -11135.982,E2 -11135.982} C_VEL
LIN {X 0,Y 397.136,Z 495.831,A -85,B 0,C 180,E1 -11139.704,E2 -11139.704} C_VEL
LIN {X 0,Y 397.179,Z 495.822,A -85,B 0,C 180,E1 -11142.845,E2 -11142.845} C_VEL
LIN {X 0,Y 397.224,Z 495.816,A -85,B 0,C 180,E1 -11146.679,E2 -11146.679} C_VEL
LIN {X 0,Y 397.226,Z 495.82,A -85,B 0,C 180,E1 -11149.809,E2 -11149.809} C_VEL
LIN {X 0,Y 397.361,Z 495.799,A -85,B 0,C 180,E1 -11152.888,E2 -11152.888} C_VEL
LIN {X 0,Y 397.253,Z 495.812,A -85,B 0,C 180,E1 -11154.925,E2 -11154.925} C_VEL
LIN {X 0,Y 397.45,Z 495.792,A -85,B 0,C 180,E1 -11157.973,E2 -11157.973} C_VEL
LIN {X 0,Y 397.578,Z 495.776,A -85,B 0,C 180,E1 -11160,E2 -11160} C_VEL
LIN {X 0,Y 397.381,Z 495.797,A -85,B 0,C 180,E1 -11163.041,E2 -11163.041} C_VEL
LIN {X 0,Y 397.361,Z 495.8,A -85,B 0,C 180,E1 -11167.112,E2 -11167.112} C_VEL
LIN {X 0,Y 397.222,Z 495.818,A -85,B 0,C 180,E1 -11170.191,E2 -11170.191} C_VEL
LIN {X 0,Y 397.223,Z 495.818,A -85,B 0,C 180,E1 -11173.321,E2 -11173.321} C_VEL
LIN {X 0,Y 397.179,Z 495.824,A -85,B 0,C 180,E1 -11177.155,E2 -11177.155} C_VEL
LIN {X 0,Y 397.1,Z 495.832,A -85,B 0,C 180,E1 -11180.73,E2 -11180.73} C_VEL
LIN {X 0,Y 397.13,Z 495.83,A -85,B 0,C 180,E1 -11184.018,E2 -11184.018} C_VEL
LIN {X 0,Y 397.192,Z 495.823,A -85,B 0,C 180,E1 -11187.39,E2 -11187.39} C_VEL
LIN {X 0,Y 397.084,Z 495.834,A -85,B 0,C 180,E1 -11190.882,E2 -11190.882} C_VEL
LIN {X 0,Y 397.123,Z 495.829,A -85,B 0,C 180,E1 -11194.493,E2 -11194.493} C_VEL
LIN {X 0,Y 397.103,Z 495.831,A -85,B 0,C 180,E1 -11198.275,E2 -11198.275} C_VEL
LIN {X 0,Y 397.086,Z 495.835,A -85,B 0,C 180,E1 -11200.909,E2 -11200.909} C_VEL
LIN {X 0,Y 397.101,Z 495.835,A -85,B 0,C 180,E1 -11203.648,E2 -11203.648} C_VEL
LIN {X 0,Y 397.102,Z 495.832,A -85,B 0,C 180,E1 -11206.521,E2 -11206.521} C_VEL
LIN {X 0,Y 397.119,Z 495.833,A -85,B 0,C 180,E1 -11209.552,E2 -11209.552} C_VEL
LIN {X 0,Y 397.099,Z 495.836,A -85,B 0,C 180,E1 -11212.79,E2 -11212.79} C_VEL
LIN {X 0,Y 397.135,Z 495.975,A -85,B 0,C 180,E1 -11213.642,E2 -11213.642} C_VEL
LIN {X 0,Y 398.08,Z 501.016,A -85,B 0,C 180,E1 -11216.075,E2 -11216.075} C_VEL
LIN {X 0,Y 398.726,Z 505.3,A -85,B 0,C 180,E1 -11218.077,E2 -11218.077} C_VEL
LIN {X 0,Y 398.273,Z 511.845,A -85,B 0,C 180,E1 -11220.97,E2 -11220.97} C_VEL
LIN {X 0,Y 397.641,Z 519.666,A -85,B 0,C 180,E1 -11224.341,E2 -11224.341} C_VEL
LIN {X 0,Y 397.081,Z 527.469,A -85,B 0,C 180,E1 -11227.634,E2 -11227.634} C_VEL
LIN {X 0,Y 396.644,Z 535.254,A -85,B 0,C 180,E1 -11230.866,E2 -11230.866} C_VEL
LIN {X 0,Y 396.249,Z 544.282,A -85,B 0,C 180,E1 -11234.572,E2 -11234.572} C_VEL
LIN {X 0,Y 396.136,Z 547.88,A -85,B 0,C 180,E1 -11236.033,E2 -11236.033} C_VEL
LIN {X 0,Y 397.166,Z 557.815,A -85,B 0,C 180,E1 -11236.398,E2 -11236.398} C_VEL
LIN {X 0,Y 398.157,Z 568.593,A -85,B 0,C 180,E1 -11236.967,E2 -11236.967} C_VEL
LIN {X 0,Y 398.308,Z 576.952,A -85,B 0,C 180,E1 -11237.539,E2 -11237.539} C_VEL
LIN {X 0,Y 397.779,Z 586.918,A -85,B 0,C 180,E1 -11238.407,E2 -11238.407} C_VEL
LIN {X 0,Y 397.348,Z 594.975,A -85,B 0,C 180,E1 -11239.298,E2 -11239.298} C_VEL
LIN {X 0,Y 396.952,Z 600.755,A -85,B 0,C 180,E1 -11240.06,E2 -11240.06} C_VEL
LIN {X 0,Y 396.585,Z 607.171,A -85,B 0,C 180,E1 -11241.08,E2 -11241.08} C_VEL
LIN {X 0,Y 396.24,Z 613.661,A -85,B 0,C 180,E1 -11242.356,E2 -11242.356} C_VEL
LIN {X 0,Y 395.952,Z 619.111,A -85,B 0,C 180,E1 -11243.709,E2 -11243.709} C_VEL
LIN {X 0,Y 395.893,Z 624.133,A -85,B 0,C 180,E1 -11245.419,E2 -11245.419} C_VEL
LIN {X 0,Y 395.798,Z 627.159,A -85,B 0,C 180,E1 -11246.947,E2 -11246.947} C_VEL
LIN {X 0,Y 395.831,Z 628.509,A -85,B 0,C 180,E1 -11247.966,E2 -11247.966} C_VEL
LIN {X 0,Y 395.828,Z 629.358,A -85,B 0,C 180,E1 -11248.983,E2 -11248.983} C_VEL
LIN {X 0,Y 395.825,Z 629.663,A -85,B 0,C 180,E1 -11250.001,E2 -11250.001} C_VEL
LIN {X 0,Y 395.828,Z 629.388,A -85,B 0,C 180,E1 -11251.018,E2 -11251.018} C_VEL
LIN {X 0,Y 395.828,Z 628.624,A -85,B 0,C 180,E1 -11252.036,E2 -11252.036} C_VEL
LIN {X 0,Y 395.785,Z 627.363,A -85,B 0,C 180,E1 -11253.054,E2 -11253.054} C_VEL
LIN {X 0,Y 395.894,Z 624.421,A -85,B 0,C 180,E1 -11254.582,E2 -11254.582} C_VEL
LIN {X 0,Y 395.922,Z 621.721,A -85,B 0,C 180,E1 -11255.603,E2 -11255.603} C_VEL
LIN {X 0,Y 396.085,Z 617.871,A -85,B 0,C 180,E1 -11256.765,E2 -11256.765} C_VEL
LIN {X 0,Y 396.387,Z 612.188,A -85,B 0,C 180,E1 -11258.155,E2 -11258.155} C_VEL
LIN {X 0,Y 396.732,Z 607.104,A -85,B 0,C 180,E1 -11259.174,E2 -11259.174} C_VEL
LIN {X 0,Y 397.191,Z 601.034,A -85,B 0,C 180,E1 -11260.192,E2 -11260.192} C_VEL
LIN {X 0,Y 397.841,Z 592.721,A -85,B 0,C 180,E1 -11261.334,E2 -11261.334} C_VEL
LIN {X 0,Y 398.48,Z 583.658,A -85,B 0,C 180,E1 -11262.349,E2 -11262.349} C_VEL
LIN {X 0,Y 399.022,Z 573.784,A -85,B 0,C 180,E1 -11263.237,E2 -11263.237} C_VEL
LIN {X 0,Y 398.592,Z 563.382,A -85,B 0,C 180,E1 -11264.003,E2 -11264.003} C_VEL
LIN {X 0,Y 397.715,Z 555.082,A -85,B 0,C 180,E1 -11264.52,E2 -11264.52} C_VEL
LIN {X 0,Y 396.151,Z 545.942,A -85,B 0,C 180,E1 -11265.038,E2 -11265.038} C_VEL
LIN {X 0,Y 396.422,Z 539.01,A -85,B 0,C 180,E1 -11268.075,E2 -11268.075} C_VEL
LIN {X 0,Y 396.809,Z 531.947,A -85,B 0,C 180,E1 -11271.29,E2 -11271.29} C_VEL
LIN {X 0,Y 397.34,Z 525.146,A -85,B 0,C 180,E1 -11274.561,E2 -11274.561} C_VEL
LIN {X 0,Y 398.019,Z 518.491,A -85,B 0,C 180,E1 -11278.009,E2 -11278.009} C_VEL
LIN {X 0,Y 398.635,Z 513.671,A -85,B 0,C 180,E1 -11280.749,E2 -11280.749} C_VEL
LIN {X 0,Y 399.053,Z 509.958,A -85,B 0,C 180,E1 -11283.091,E2 -11283.091} C_VEL
LIN {X 0,Y 399.111,Z 508.237,A -85,B 0,C 180,E1 -11284.298,E2 -11284.298} C_VEL
LIN {X 0,Y 398.734,Z 505.15,A -85,B 0,C 180,E1 -11286.819,E2 -11286.819} C_VEL
LIN {X 0,Y 398.297,Z 502.56,A -85,B 0,C 180,E1 -11289.437,E2 -11289.437} C_VEL
LIN {X 0,Y 397.939,Z 500.526,A -85,B 0,C 180,E1 -11292.154,E2 -11292.154} C_VEL
LIN {X 0,Y 397.691,Z 499.128,A -85,B 0,C 180,E1 -11295.018,E2 -11295.018} C_VEL
LIN {X 0,Y 397.56,Z 498.435,A -85,B 0,C 180,E1 -11297.943,E2 -11297.943} C_VEL
LIN {X 0,Y 397.549,Z 498.468,A -85,B 0,C 180,E1 -11301.065,E2 -11301.065} C_VEL
LIN {X 0,Y 397.636,Z 499.25,A -85,B 0,C 180,E1 -11304.393,E2 -11304.393} C_VEL
LIN {X 0,Y 397.702,Z 500.24,A -85,B 0,C 180,E1 -11306.783,E2 -11306.783} C_VEL
LIN {X 0,Y 397.567,Z 501.537,A -85,B 0,C 180,E1 -11309.16,E2 -11309.16} C_VEL
LIN {X 0,Y 397.207,Z 503.863,A -85,B 0,C 180,E1 -11312.611,E2 -11312.611} C_VEL
LIN {X 0,Y 396.885,Z 506.5,A -85,B 0,C 180,E1 -11315.966,E2 -11315.966} C_VEL
LIN {X 0,Y 396.693,Z 509.343,A -85,B 0,C 180,E1 -11319.248,E2 -11319.248} C_VEL
LIN {X 0,Y 396.492,Z 512.36,A -85,B 0,C 180,E1 -11322.462,E2 -11322.462} C_VEL
LIN {X 0,Y 396.392,Z 515.23,A -85,B 0,C 180,E1 -11325.152,E2 -11325.152} C_VEL
LIN {X 0,Y 399.253,Z 525.983,A -85,B 0,C 180,E1 -11325.874,E2 -11325.874} C_VEL
LIN {X 0,Y 400.409,Z 532.169,A -85,B 0,C 180,E1 -11326.336,E2 -11326.336} C_VEL
LIN {X 0,Y 399.805,Z 542.739,A -85,B 0,C 180,E1 -11327.178,E2 -11327.178} C_VEL
LIN {X 0,Y 399.249,Z 550.422,A -85,B 0,C 180,E1 -11327.934,E2 -11327.934} C_VEL
LIN {X 0,Y 398.678,Z 557.855,A -85,B 0,C 180,E1 -11328.819,E2 -11328.819} C_VEL
LIN {X 0,Y 398.081,Z 564.924,A -85,B 0,C 180,E1 -11329.831,E2 -11329.831} C_VEL
LIN {X 0,Y 397.521,Z 572.178,A -85,B 0,C 180,E1 -11331.101,E2 -11331.101} C_VEL
LIN {X 0,Y 397.017,Z 578.76,A -85,B 0,C 180,E1 -11332.604,E2 -11332.604} C_VEL
LIN {X 0,Y 396.474,Z 583.172,A -85,B 0,C 180,E1 -11333.895,E2 -11333.895} C_VEL
LIN {X 0,Y 396.381,Z 587.026,A -85,B 0,C 180,E1 -11335.424,E2 -11335.424} C_VEL
LIN {X 0,Y 396.097,Z 589.653,A -85,B 0,C 180,E1 -11336.949,E2 -11336.949} C_VEL
LIN {X 0,Y 395.966,Z 590.653,A -85,B 0,C 180,E1 -11337.966,E2 -11337.966} C_VEL
LIN {X 0,Y 395.859,Z 591.167,A -85,B 0,C 180,E1 -11338.983,E2 -11338.983} C_VEL
LIN {X 0,Y 395.828,Z 591.202,A -85,B 0,C 180,E1 -11340,E2 -11340} C_VEL
LIN {X 0,Y 395.846,Z 590.743,A -85,B 0,C 180,E1 -11341.017,E2 -11341.017} C_VEL
LIN {X 0,Y 395.938,Z 589.689,A -85,B 0,C 180,E1 -11342.035,E2 -11342.035} C_VEL
LIN {X 0,Y 396.009,Z 587.154,A -85,B 0,C 180,E1 -11343.561,E2 -11343.561} C_VEL
LIN {X 0,Y 396.137,Z 583.244,A -85,B 0,C 180,E1 -11345.089,E2 -11345.089} C_VEL
LIN {X 0,Y 396.43,Z 577.995,A -85,B 0,C 180,E1 -11346.6,E2 -11346.6} C_VEL
LIN {X 0,Y 396.681,Z 572.241,A -85,B 0,C 180,E1 -11347.892,E2 -11347.892} C_VEL
LIN {X 0,Y 397.064,Z 565.077,A -85,B 0,C 180,E1 -11349.166,E2 -11349.166} C_VEL
LIN {X 0,Y 397.517,Z 556.942,A -85,B 0,C 180,E1 -11350.312,E2 -11350.312} C_VEL
LIN {X 0,Y 397.982,Z 549.249,A -85,B 0,C 180,E1 -11351.201,E2 -11351.201} C_VEL
LIN {X 0,Y 398.338,Z 541.253,A -85,B 0,C 180,E1 -11351.965,E2 -11351.965} C_VEL
LIN {X 0,Y 398.856,Z 530.742,A -85,B 0,C 180,E1 -11352.768,E2 -11352.768} C_VEL
LIN {X 0,Y 397.301,Z 519.866,A -85,B 0,C 180,E1 -11353.427,E2 -11353.427} C_VEL
LIN {X 0,Y 396.041,Z 512.07,A -85,B 0,C 180,E1 -11353.809,E2 -11353.809} C_VEL
LIN {X 0,Y 396.06,Z 508.368,A -85,B 0,C 180,E1 -11356.619,E2 -11356.619} C_VEL
LIN {X 0,Y 396.131,Z 504.127,A -85,B 0,C 180,E1 -11359.896,E2 -11359.896} C_VEL
LIN {X 0,Y 396.226,Z 500.233,A -85,B 0,C 180,E1 -11362.968,E2 -11362.968} C_VEL
LIN {X 0,Y 396.449,Z 496.1,A -85,B 0,C 180,E1 -11366.378,E2 -11366.378} C_VEL
LIN {X 0,Y 396.907,Z 498.866,A -85,B 0,C 180,E1 -11367.705,E2 -11367.705} C_VEL
LIN {X 0,Y 396.768,Z 505.68,A -85,B 0,C 180,E1 -11370.909,E2 -11370.909} C_VEL
LIN {X 0,Y 396.663,Z 511.368,A -85,B 0,C 180,E1 -11373.618,E2 -11373.618} C_VEL
LIN {X 0,Y 396.462,Z 518.61,A -85,B 0,C 180,E1 -11377.088,E2 -11377.088} C_VEL
LIN {X 0,Y 396.259,Z 525.285,A -85,B 0,C 180,E1 -11380.302,E2 -11380.302} C_VEL
LIN {X 0,Y 396.252,Z 528.076,A -85,B 0,C 180,E1 -11381.647,E2 -11381.647} C_VEL
LIN {X 0,Y 398.112,Z 537.882,A -85,B 0,C 180,E1 -11382.093,E2 -11382.093} C_VEL
LIN {X 0,Y 399.533,Z 548.666,A -85,B 0,C 180,E1 -11382.734,E2 -11382.734} C_VEL
LIN {X 0,Y 398.924,Z 559.709,A -85,B 0,C 180,E1 -11383.559,E2 -11383.559} C_VEL
LIN {X 0,Y 398.438,Z 568.208,A -85,B 0,C 180,E1 -11384.381,E2 -11384.381} C_VEL
LIN {X 0,Y 397.823,Z 576.656,A -85,B 0,C 180,E1 -11385.393,E2 -11385.393} C_VEL
LIN {X 0,Y 397.297,Z 584.055,A -85,B 0,C 180,E1 -11386.491,E2 -11386.491} C_VEL
LIN {X 0,Y 396.803,Z 590.531,A -85,B 0,C 180,E1 -11387.697,E2 -11387.697} C_VEL
LIN {X 0,Y 396.421,Z 596.082,A -85,B 0,C 180,E1 -11389.007,E2 -11389.007} C_VEL
LIN {X 0,Y 396.136,Z 600.417,A -85,B 0,C 180,E1 -11390.305,E2 -11390.305} C_VEL
LIN {X 0,Y 395.952,Z 603.7,A -85,B 0,C 180,E1 -11391.593,E2 -11391.593} C_VEL
LIN {X 0,Y 395.739,Z 606.333,A -85,B 0,C 180,E1 -11393.05,E2 -11393.05} C_VEL
LIN {X 0,Y 395.624,Z 608.093,A -85,B 0,C 180,E1 -11394.802,E2 -11394.802} C_VEL
LIN {X 0,Y 395.59,Z 608.231,A -85,B 0,C 180,E1 -11396.616,E2 -11396.616} C_VEL
LIN {X 0,Y 395.68,Z 606.834,A -85,B 0,C 180,E1 -11398.492,E2 -11398.492} C_VEL
LIN {X 0,Y 395.884,Z 603.903,A -85,B 0,C 180,E1 -11400.193,E2 -11400.193} C_VEL
LIN {X 0,Y 396.016,Z 601.006,A -85,B 0,C 180,E1 -11401.369,E2 -11401.369} C_VEL
LIN {X 0,Y 396.342,Z 596.204,A -85,B 0,C 180,E1 -11402.831,E2 -11402.831} C_VEL
LIN {X 0,Y 396.721,Z 590.454,A -85,B 0,C 180,E1 -11404.188,E2 -11404.188} C_VEL
LIN {X 0,Y 397.138,Z 583.789,A -85,B 0,C 180,E1 -11405.425,E2 -11405.425} C_VEL
LIN {X 0,Y 397.552,Z 577.134,A -85,B 0,C 180,E1 -11406.422,E2 -11406.422} C_VEL
LIN {X 0,Y 398.092,Z 568.919,A -85,B 0,C 180,E1 -11407.419,E2 -11407.419} C_VEL
LIN {X 0,Y 398.478,Z 561.887,A -85,B 0,C 180,E1 -11408.124,E2 -11408.124} C_VEL
LIN {X 0,Y 399.006,Z 553.128,A -85,B 0,C 180,E1 -11408.833,E2 -11408.833} C_VEL
LIN {X 0,Y 399.1,Z 547.304,A -85,B 0,C 180,E1 -11409.23,E2 -11409.23} C_VEL
LIN {X 0,Y 397.602,Z 537.142,A -85,B 0,C 180,E1 -11409.816,E2 -11409.816} C_VEL
LIN {X 0,Y 396.047,Z 528.081,A -85,B 0,C 180,E1 -11410.221,E2 -11410.221} C_VEL
LIN {X 0,Y 396.181,Z 520.715,A -85,B 0,C 180,E1 -11414.04,E2 -11414.04} C_VEL
LIN {X 0,Y 396.394,Z 513.622,A -85,B 0,C 180,E1 -11417.715,E2 -11417.715} C_VEL
LIN {X 0,Y 396.545,Z 507.683,A -85,B 0,C 180,E1 -11420.821,E2 -11420.821} C_VEL
LIN {X 0,Y 396.701,Z 500.675,A -85,B 0,C 180,E1 -11424.408,E2 -11424.408} C_VEL
LIN {X 0,Y 396.806,Z 495.873,A -85,B 0,C 180,E1 -11426.954,E2 -11426.954} C_VEL
LIN {X 0,Y 397.57,Z 495.776,A -85,B 0,C 180,E1 -11429.999,E2 -11429.999} C_VEL
LIN {X 0,Y 397.382,Z 495.797,A -85,B 0,C 180,E1 -11433.041,E2 -11433.041} C_VEL
LIN {X 0,Y 397.366,Z 495.799,A -85,B 0,C 180,E1 -11437.111,E2 -11437.111} C_VEL
LIN {X 0,Y 397.218,Z 495.821,A -85,B 0,C 180,E1 -11440.19,E2 -11440.19} C_VEL
LIN {X 0,Y 397.201,Z 495.821,A -85,B 0,C 180,E1 -11440.447,E2 -11440.447} C_VEL
LIN {X 0,Y 396.514,Z 495.905,A -85,B 0,C 180,E1 -11441.294,E2 -11441.294} C_VEL
LIN {X 0,Y 393.662,Z 496.262,A -85,B 0,C 180,E1 -11442.671,E2 -11442.671} C_VEL
LIN {X 0,Y 391.256,Z 496.563,A -85,B 0,C 180,E1 -11443.784,E2 -11443.784} C_VEL
LIN {X 0,Y 390.217,Z 496.691,A -85,B 0,C 180,E1 -11444.644,E2 -11444.644} C_VEL
LIN {X 0,Y 390.129,Z 496.7,A -85,B 0,C 180,E1 -11444.935,E2 -11444.935} C_VEL
LIN {X 0,Y 390.129,Z 496.702,A -85,B 0,C 180,E1 -11447.833,E2 -11447.833} C_VEL
LIN {X 0,Y 390.056,Z 496.708,A -85,B 0,C 180,E1 -11451.122,E2 -11451.122} C_VEL
LIN {X 0,Y 390.08,Z 496.709,A -85,B 0,C 180,E1 -11454.48,E2 -11454.48} C_VEL
LIN {X 0,Y 390.115,Z 496.706,A -85,B 0,C 180,E1 -11458.025,E2 -11458.025} C_VEL
LIN {X 0,Y 390.027,Z 496.714,A -85,B 0,C 180,E1 -11461.503,E2 -11461.503} C_VEL
LIN {X 0,Y 390.067,Z 496.712,A -85,B 0,C 180,E1 -11464.024,E2 -11464.024} C_VEL
LIN {X 0,Y 390.045,Z 496.712,A -85,B 0,C 180,E1 -11467.551,E2 -11467.551} C_VEL
LIN {X 0,Y 390.056,Z 496.709,A -85,B 0,C 180,E1 -11470.821,E2 -11470.821} C_VEL
LIN {X 0,Y 390.06,Z 496.712,A -85,B 0,C 180,E1 -11473.887,E2 -11473.887} C_VEL
LIN {X 0,Y 390.116,Z 496.702,A -85,B 0,C 180,E1 -11476.798,E2 -11476.798} C_VEL
LIN {X 0,Y 390.076,Z 496.709,A -85,B 0,C 180,E1 -11479.563,E2 -11479.563} C_VEL
LIN {X 0,Y 390.045,Z 496.712,A -85,B 0,C 180,E1 -11482.448,E2 -11482.448} C_VEL
LIN {X 0,Y 390.065,Z 496.712,A -85,B 0,C 180,E1 -11486.045,E2 -11486.045} C_VEL
LIN {X 0,Y 390.044,Z 496.715,A -85,B 0,C 180,E1 -11489.869,E2 -11489.869} C_VEL
LIN {X 0,Y 390.111,Z 496.703,A -85,B 0,C 180,E1 -11493.232,E2 -11493.232} C_VEL
LIN {X 0,Y 390.104,Z 496.703,A -85,B 0,C 180,E1 -11496.75,E2 -11496.75} C_VEL
LIN {X 0,Y 390.101,Z 496.708,A -85,B 0,C 180,E1 -11499.983,E2 -11499.983} C_VEL
LIN {X 0,Y 390.135,Z 496.7,A -85,B 0,C 180,E1 -11503.248,E2 -11503.248} C_VEL
LIN {X 0,Y 390.192,Z 496.692,A -85,B 0,C 180,E1 -11506.561,E2 -11506.561} C_VEL
LIN {X 0,Y 390.176,Z 496.697,A -85,B 0,C 180,E1 -11509.623,E2 -11509.623} C_VEL
LIN {X 0,Y 390.316,Z 496.676,A -85,B 0,C 180,E1 -11512.759,E2 -11512.759} C_VEL
LIN {X 0,Y 390.225,Z 496.688,A -85,B 0,C 180,E1 -11514.833,E2 -11514.833} C_VEL
LIN {X 0,Y 390.418,Z 496.668,A -85,B 0,C 180,E1 -11517.937,E2 -11517.937} C_VEL
LIN {X 0,Y 390.548,Z 496.652,A -85,B 0,C 180,E1 -11520,E2 -11520} C_VEL
LIN {X 0,Y 390.315,Z 496.678,A -85,B 0,C 180,E1 -11523.096,E2 -11523.096} C_VEL
LIN {X 0,Y 390.328,Z 496.677,A -85,B 0,C 180,E1 -11526.202,E2 -11526.202} C_VEL
LIN {X 0,Y 390.312,Z 496.679,A -85,B 0,C 180,E1 -11528.282,E2 -11528.282} C_VEL
LIN {X 0,Y 390.168,Z 496.695,A -85,B 0,C 180,E1 -11532.483,E2 -11532.483} C_VEL
LIN {X 0,Y 390.136,Z 496.704,A -85,B 0,C 180,E1 -11535.677,E2 -11535.677} C_VEL
LIN {X 0,Y 390.103,Z 496.703,A -85,B 0,C 180,E1 -11538.922,E2 -11538.922} C_VEL
LIN {X 0,Y 390.037,Z 496.713,A -85,B 0,C 180,E1 -11542.234,E2 -11542.234} C_VEL
LIN {X 0,Y 390.116,Z 496.705,A -85,B 0,C 180,E1 -11545.744,E2 -11545.744} C_VEL
LIN {X 0,Y 390.063,Z 496.71,A -85,B 0,C 180,E1 -11549.109,E2 -11549.109} C_VEL
LIN {X 0,Y 390.053,Z 496.709,A -85,B 0,C 180,E1 -11552.72,E2 -11552.72} C_VEL
LIN {X 0,Y 390.054,Z 496.712,A -85,B 0,C 180,E1 -11555.826,E2 -11555.826} C_VEL
LIN {X 0,Y 390.068,Z 496.71,A -85,B 0,C 180,E1 -11559.219,E2 -11559.219} C_VEL
LIN {X 0,Y 390.042,Z 496.711,A -85,B 0,C 180,E1 -11562.375,E2 -11562.375} C_VEL
LIN {X 0,Y 390.043,Z 496.715,A -85,B 0,C 180,E1 -11565.355,E2 -11565.355} C_VEL
LIN {X 0,Y 390.066,Z 496.708,A -85,B 0,C 180,E1 -11568.192,E2 -11568.192} C_VEL
LIN {X 0,Y 390.093,Z 496.705,A -85,B 0,C 180,E1 -11570.909,E2 -11570.909} C_VEL
LIN {X 0,Y 390.111,Z 496.765,A -85,B 0,C 180,E1 -11573.443,E2 -11573.443} C_VEL
LIN {X 0,Y 391.329,Z 503.594,A -85,B 0,C 180,E1 -11576.787,E2 -11576.787} C_VEL
LIN {X 0,Y 391.669,Z 507.562,A -85,B 0,C 180,E1 -11578.644,E2 -11578.644} C_VEL
LIN {X 0,Y 390.982,Z 515.385,A -85,B 0,C 180,E1 -11582.138,E2 -11582.138} C_VEL
LIN {X 0,Y 390.334,Z 523.184,A -85,B 0,C 180,E1 -11585.537,E2 -11585.537} C_VEL
LIN {X 0,Y 389.816,Z 530.949,A -85,B 0,C 180,E1 -11588.865,E2 -11588.865} C_VEL
LIN {X 0,Y 389.356,Z 540.108,A -85,B 0,C 180,E1 -11592.727,E2 -11592.727} C_VEL
LIN {X 0,Y 389.044,Z 547.555,A -85,B 0,C 180,E1 -11595.792,E2 -11595.792} C_VEL
LIN {X 0,Y 390.142,Z 557.394,A -85,B 0,C 180,E1 -11596.16,E2 -11596.16} C_VEL
LIN {X 0,Y 391.034,Z 567.449,A -85,B 0,C 180,E1 -11596.691,E2 -11596.691} C_VEL
LIN {X 0,Y 391.418,Z 575.127,A -85,B 0,C 180,E1 -11597.216,E2 -11597.216} C_VEL
LIN {X 0,Y 390.912,Z 585.323,A -85,B 0,C 180,E1 -11598.068,E2 -11598.068} C_VEL
LIN {X 0,Y 390.425,Z 593.635,A -85,B 0,C 180,E1 -11598.974,E2 -11598.974} C_VEL
LIN {X 0,Y 389.95,Z 600.457,A -85,B 0,C 180,E1 -11599.88,E2 -11599.88} C_VEL
LIN {X 0,Y 389.536,Z 606.891,A -85,B 0,C 180,E1 -11600.917,E2 -11600.917} C_VEL
LIN {X 0,Y 389.254,Z 612.224,A -85,B 0,C 180,E1 -11601.957,E2 -11601.957} C_VEL
LIN {X 0,Y 389.016,Z 616.753,A -85,B 0,C 180,E1 -11603.022,E2 -11603.022} C_VEL
LIN {X 0,Y 388.83,Z 620.502,A -85,B 0,C 180,E1 -11604.095,E2 -11604.095} C_VEL
LIN {X 0,Y 388.823,Z 623.908,A -85,B 0,C 180,E1 -11605.335,E2 -11605.335} C_VEL
LIN {X 0,Y 388.702,Z 626.943,A -85,B 0,C 180,E1 -11606.891,E2 -11606.891} C_VEL
LIN {X 0,Y 388.729,Z 628.303,A -85,B 0,C 180,E1 -11607.928,E2 -11607.928} C_VEL
LIN {X 0,Y 388.757,Z 629.163,A -85,B 0,C 180,E1 -11608.965,E2 -11608.965} C_VEL
LIN {X 0,Y 388.752,Z 629.469,A -85,B 0,C 180,E1 -11610.001,E2 -11610.001} C_VEL
LIN {X 0,Y 388.757,Z 629.202,A -85,B 0,C 180,E1 -11611.036,E2 -11611.036} C_VEL
LIN {X 0,Y 388.725,Z 628.446,A -85,B 0,C 180,E1 -11612.073,E2 -11612.073} C_VEL
LIN {X 0,Y 388.69,Z 627.195,A -85,B 0,C 180,E1 -11613.11,E2 -11613.11} C_VEL
LIN {X 0,Y 388.825,Z 624.266,A -85,B 0,C 180,E1 -11614.666,E2 -11614.666} C_VEL
LIN {X 0,Y 388.856,Z 620.887,A -85,B 0,C 180,E1 -11615.941,E2 -11615.941} C_VEL
LIN {X 0,Y 389.095,Z 616.388,A -85,B 0,C 180,E1 -11617.264,E2 -11617.264} C_VEL
LIN {X 0,Y 389.431,Z 610.967,A -85,B 0,C 180,E1 -11618.563,E2 -11618.563} C_VEL
LIN {X 0,Y 389.949,Z 604.264,A -85,B 0,C 180,E1 -11619.859,E2 -11619.859} C_VEL
LIN {X 0,Y 390.621,Z 596.037,A -85,B 0,C 180,E1 -11621.153,E2 -11621.153} C_VEL
LIN {X 0,Y 391.34,Z 586.578,A -85,B 0,C 180,E1 -11622.314,E2 -11622.314} C_VEL
LIN {X 0,Y 392.004,Z 578.925,A -85,B 0,C 180,E1 -11623.083,E2 -11623.083} C_VEL
LIN {X 0,Y 392.091,Z 571.746,A -85,B 0,C 180,E1 -11623.711,E2 -11623.711} C_VEL
LIN {X 0,Y 391.734,Z 563.205,A -85,B 0,C 180,E1 -11624.35,E2 -11624.35} C_VEL
LIN {X 0,Y 390.501,Z 553.183,A -85,B 0,C 180,E1 -11624.994,E2 -11624.994} C_VEL
LIN {X 0,Y 389.121,Z 545.527,A -85,B 0,C 180,E1 -11625.451,E2 -11625.451} C_VEL
LIN {X 0,Y 389.382,Z 538.948,A -85,B 0,C 180,E1 -11628.413,E2 -11628.413} C_VEL
LIN {X 0,Y 389.751,Z 533.106,A -85,B 0,C 180,E1 -11631.14,E2 -11631.14} C_VEL
LIN {X 0,Y 390.303,Z 526.346,A -85,B 0,C 180,E1 -11634.466,E2 -11634.466} C_VEL
LIN {X 0,Y 391.055,Z 519.186,A -85,B 0,C 180,E1 -11638.283,E2 -11638.283} C_VEL
LIN {X 0,Y 391.772,Z 514.004,A -85,B 0,C 180,E1 -11641.348,E2 -11641.348} C_VEL
LIN {X 0,Y 392.14,Z 510.424,A -85,B 0,C 180,E1 -11643.752,E2 -11643.752} C_VEL
LIN {X 0,Y 391.895,Z 507.252,A -85,B 0,C 180,E1 -11646.286,E2 -11646.286} C_VEL
LIN {X 0,Y 391.39,Z 504.111,A -85,B 0,C 180,E1 -11649.455,E2 -11649.455} C_VEL
LIN {X 0,Y 390.976,Z 501.911,A -85,B 0,C 180,E1 -11652.524,E2 -11652.524} C_VEL
LIN {X 0,Y 390.713,Z 500.405,A -85,B 0,C 180,E1 -11656.014,E2 -11656.014} C_VEL
LIN {X 0,Y 390.627,Z 499.917,A -85,B 0,C 180,E1 -11659.083,E2 -11659.083} C_VEL
LIN {X 0,Y 390.623,Z 500.171,A -85,B 0,C 180,E1 -11662.34,E2 -11662.34} C_VEL
LIN {X 0,Y 390.75,Z 501.203,A -85,B 0,C 180,E1 -11665.829,E2 -11665.829} C_VEL
LIN {X 0,Y 390.637,Z 502.495,A -85,B 0,C 180,E1 -11668.551,E2 -11668.551} C_VEL
LIN {X 0,Y 390.274,Z 504.704,A -85,B 0,C 180,E1 -11672.082,E2 -11672.082} C_VEL
LIN {X 0,Y 389.921,Z 507.251,A -85,B 0,C 180,E1 -11675.509,E2 -11675.509} C_VEL
LIN {X 0,Y 389.676,Z 510.036,A -85,B 0,C 180,E1 -11678.856,E2 -11678.856} C_VEL
LIN {X 0,Y 389.477,Z 513.012,A -85,B 0,C 180,E1 -11682.136,E2 -11682.136} C_VEL
LIN {X 0,Y 389.337,Z 515.492,A -85,B 0,C 180,E1 -11684.714,E2 -11684.714} C_VEL
LIN {X 0,Y 392.249,Z 526.121,A -85,B 0,C 180,E1 -11685.473,E2 -11685.473} C_VEL
LIN {X 0,Y 393.627,Z 533.23,A -85,B 0,C 180,E1 -11686.037,E2 -11686.037} C_VEL
LIN {X 0,Y 393.105,Z 542.873,A -85,B 0,C 180,E1 -11686.824,E2 -11686.824} C_VEL
LIN {X 0,Y 392.414,Z 551.745,A -85,B 0,C 180,E1 -11687.721,E2 -11687.721} C_VEL
LIN {X 0,Y 391.829,Z 559.028,A -85,B 0,C 180,E1 -11688.621,E2 -11688.621} C_VEL
LIN {X 0,Y 391.096,Z 567.551,A -85,B 0,C 180,E1 -11689.909,E2 -11689.909} C_VEL
LIN {X 0,Y 390.444,Z 574.207,A -85,B 0,C 180,E1 -11691.199,E2 -11691.199} C_VEL
LIN {X 0,Y 390.12,Z 578.605,A -85,B 0,C 180,E1 -11692.235,E2 -11692.235} C_VEL
LIN {X 0,Y 389.691,Z 582.296,A -85,B 0,C 180,E1 -11693.268,E2 -11693.268} C_VEL
LIN {X 0,Y 389.367,Z 586.478,A -85,B 0,C 180,E1 -11694.822,E2 -11694.822} C_VEL
LIN {X 0,Y 389.268,Z 588.596,A -85,B 0,C 180,E1 -11695.859,E2 -11695.859} C_VEL
LIN {X 0,Y 389.045,Z 590.154,A -85,B 0,C 180,E1 -11696.893,E2 -11696.893} C_VEL
LIN {X 0,Y 388.901,Z 591.107,A -85,B 0,C 180,E1 -11697.929,E2 -11697.929} C_VEL
LIN {X 0,Y 388.789,Z 591.564,A -85,B 0,C 180,E1 -11698.964,E2 -11698.964} C_VEL
LIN {X 0,Y 388.755,Z 591.535,A -85,B 0,C 180,E1 -11700,E2 -11700} C_VEL
LIN {X 0,Y 388.776,Z 591.022,A -85,B 0,C 180,E1 -11701.036,E2 -11701.036} C_VEL
LIN {X 0,Y 388.872,Z 589.952,A -85,B 0,C 180,E1 -11702.072,E2 -11702.072} C_VEL
LIN {X 0,Y 388.914,Z 587.308,A -85,B 0,C 180,E1 -11703.626,E2 -11703.626} C_VEL
LIN {X 0,Y 389.009,Z 584.868,A -85,B 0,C 180,E1 -11704.663,E2 -11704.663} C_VEL
LIN {X 0,Y 389.223,Z 579.921,A -85,B 0,C 180,E1 -11706.22,E2 -11706.22} C_VEL
LIN {X 0,Y 389.516,Z 575.8,A -85,B 0,C 180,E1 -11707.256,E2 -11707.256} C_VEL
LIN {X 0,Y 389.765,Z 569.389,A -85,B 0,C 180,E1 -11708.555,E2 -11708.555} C_VEL
LIN {X 0,Y 390.151,Z 563.14,A -85,B 0,C 180,E1 -11709.592,E2 -11709.592} C_VEL
LIN {X 0,Y 390.59,Z 555.596,A -85,B 0,C 180,E1 -11710.628,E2 -11710.628} C_VEL
LIN {X 0,Y 391.138,Z 546.371,A -85,B 0,C 180,E1 -11711.662,E2 -11711.662} C_VEL
LIN {X 0,Y 391.63,Z 536.275,A -85,B 0,C 180,E1 -11712.538,E2 -11712.538} C_VEL
LIN {X 0,Y 391.683,Z 529.173,A -85,B 0,C 180,E1 -11713.047,E2 -11713.047} C_VEL
LIN {X 0,Y 389.829,Z 518.003,A -85,B 0,C 180,E1 -11713.704,E2 -11713.704} C_VEL
LIN {X 0,Y 388.951,Z 512.339,A -85,B 0,C 180,E1 -11714.005,E2 -11714.005} C_VEL
LIN {X 0,Y 388.998,Z 508.688,A -85,B 0,C 180,E1 -11716.802,E2 -11716.802} C_VEL
